   1:  PR[GP1:91,2] = PR[GP1:90,2] + -13.749;
   1:L PR[91] R[100]mm/sec CNT100;
   1:  PR[GP1:91,1] = PR[GP1:90,1] + -6.828;
   1:  PR[GP1:91,2] = PR[GP1:90,2] + -9.017;
   1:L PR[91] R[100]mm/sec CNT100;
   1:  PR[GP1:91,1] = PR[GP1:90,1] + -5.853;
   1:  PR[GP1:91,2] = PR[GP1:90,2] + -5.100;
   1:L PR[91] R[100]mm/sec CNT100;
   1:  PR[GP1:91,1] = PR[GP1:90,1] + -4.023;
   1:  PR[GP1:91,2] = PR[GP1:90,2] + -1.796;
   1:L PR[91] R[100]mm/sec CNT100;
   1:  PR[GP1:91,1] = PR[GP1:90,1] + -0.454;
   1:  PR[GP1:91,2] = PR[GP1:90,2] + -0.472;
   1:L PR[91] R[100]mm/sec CNT100;
   1:  PR[GP1:91,1] = PR[GP1:90,1] + 0.667;
   1:L PR[91] R[100]mm/sec CNT100;
   1:  PR[GP1:91,1] = PR[GP1:90,1] + 4.236;
   1:  PR[GP1:91,2] = PR[GP1:90,2] + -1.796;
   1:L PR[91] R[100]mm/sec CNT100;
   1:  PR[GP1:91,1] = PR[GP1:90,1] + 6.052;
   1:  PR[GP1:91,2] = PR[GP1:90,2] + -5.076;
   1:L PR[91] R[100]mm/sec CNT100;
   1:  PR[GP1:91,1] = PR[GP1:90,1] + 7.757;
   1:  PR[GP1:91,2] = PR[GP1:90,2] + -9.935;
   1:L PR[91] R[100]mm/sec CNT100;
   1:  PR[GP1:91,1] = PR[GP1:90,1] + 8.713;
   1:  PR[GP1:91,2] = PR[GP1:90,2] + -13.775;
   1:L PR[91] R[100]mm/sec CNT100;
   1:  PR[GP1:91,1] = PR[GP1:90,1] + 10.319;
   1:  PR[GP1:91,2] = PR[GP1:90,2] + -17.268;
   1:L PR[91] R[100]mm/sec CNT100;
   1:  PR[GP1:91,1] = PR[GP1:90,1] + 13.595;
   1:  PR[GP1:91,2] = PR[GP1:90,2] + -21.070;
   1:L PR[91] R[100]mm/sec CNT100;
   1:  PR[GP1:91,1] = PR[GP1:90,1] + 15.888;
   1:  PR[GP1:91,2] = PR[GP1:90,2] + -24.295;
   1:L PR[91] R[100]mm/sec CNT100;
   1:  PR[GP1:91,1] = PR[GP1:90,1] + 18.658;
   1:  PR[GP1:91,2] = PR[GP1:90,2] + -26.960;
   1:L PR[91] R[100]mm/sec CNT100;
   1:  PR[GP1:91,1] = PR[GP1:90,1] + 23.094;
   1:  PR[GP1:91,2] = PR[GP1:90,2] + -29.301;
   1:L PR[91] R[100]mm/sec CNT100;
   1:  PR[GP1:91,1] = PR[GP1:90,1] + 26.406;
   1:  PR[GP1:91,2] = PR[GP1:90,2] + -31.467;
   1:L PR[91] R[100]mm/sec CNT100;
   1:  PR[GP1:91,1] = PR[GP1:90,1] + 29.959;
   1:  PR[GP1:91,2] = PR[GP1:90,2] + -32.936;
   1:L PR[91] R[100]mm/sec CNT100;
   1:  PR[GP1:91,1] = PR[GP1:90,1] + 34.945;
   1:  PR[GP1:91,2] = PR[GP1:90,2] + -33.495;
   1:L PR[91] R[100]mm/sec CNT100;
   1:  PR[GP1:91,1] = PR[GP1:90,1] + 38.819;
   1:  PR[GP1:91,2] = PR[GP1:90,2] + -34.301;
   1:L PR[91] R[100]mm/sec CNT100;
   1:  PR[GP1:91,1] = PR[GP1:90,1] + 42.663;
   1:  PR[GP1:91,2] = PR[GP1:90,2] + -34.371;
   1:L PR[91] R[100]mm/sec CNT100;
   1:  PR[GP1:91,1] = PR[GP1:90,1] + 47.510;
   1:  PR[GP1:91,2] = PR[GP1:90,2] + -33.071;
   1:L PR[91] R[100]mm/sec CNT100;
   1:  PR[GP1:91,1] = PR[GP1:90,1] + 51.411;
   1:  PR[GP1:91,2] = PR[GP1:90,2] + -32.407;
   1:L PR[91] R[100]mm/sec CNT100;
   1:  PR[GP1:91,1] = PR[GP1:90,1] + 55.014;
   1:  PR[GP1:91,2] = PR[GP1:90,2] + -31.068;
   1:L PR[91] R[100]mm/sec CNT100;
   1:  PR[GP1:91,1] = PR[GP1:90,1] + 59.050;
   1:  PR[GP1:91,2] = PR[GP1:90,2] + -28.089;
   1:L PR[91] R[100]mm/sec CNT100;
   1:  PR[GP1:91,1] = PR[GP1:90,1] + 62.438;
   1:  PR[GP1:91,2] = PR[GP1:90,2] + -26.045;
   1:L PR[91] R[100]mm/sec CNT100;
   1:  PR[GP1:91,1] = PR[GP1:90,1] + 65.304;
   1:  PR[GP1:91,2] = PR[GP1:90,2] + -23.483;
   1:L PR[91] R[100]mm/sec CNT100;
   1:  PR[GP1:91,1] = PR[GP1:90,1] + 67.974;
   1:  PR[GP1:91,2] = PR[GP1:90,2] + -19.233;
   1:L PR[91] R[100]mm/sec CNT100;
   1:  PR[GP1:91,1] = PR[GP1:90,1] + 70.383;
   1:  PR[GP1:91,2] = PR[GP1:90,2] + -16.093;
   1:L PR[91] R[100]mm/sec CNT100;
   1:  PR[GP1:91,1] = PR[GP1:90,1] + 72.115;
   1:  PR[GP1:91,2] = PR[GP1:90,2] + -12.661;
   1:L PR[91] R[100]mm/sec CNT100;
   1:  PR[GP1:91,1] = PR[GP1:90,1] + 73.047;
   1:  PR[GP1:91,2] = PR[GP1:90,2] + -7.730;
   1:L PR[91] R[100]mm/sec CNT100;
   1:  PR[GP1:91,1] = PR[GP1:90,1] + 74.143;
   1:  PR[GP1:91,2] = PR[GP1:90,2] + -3.928;
   1:L PR[91] R[100]mm/sec CNT100;
   1:  PR[GP1:91,1] = PR[GP1:90,1] + 74.501;
   1:  PR[GP1:91,2] = PR[GP1:90,2] + -0.100;
   1:L PR[91] R[100]mm/sec CNT100;
   1:  PR[GP1:91,1] = PR[GP1:90,1] + 73.568;
   1:  PR[GP1:91,2] = PR[GP1:90,2] + 4.830;
   1:L PR[91] R[100]mm/sec CNT100;
   1:  PR[GP1:91,1] = PR[GP1:90,1] + 73.199;
   1:  PR[GP1:91,2] = PR[GP1:90,2] + 8.770;
   1:L PR[91] R[100]mm/sec CNT100;
   1:  PR[GP1:91,1] = PR[GP1:90,1] + 72.127;
   1:  PR[GP1:91,2] = PR[GP1:90,2] + 12.491;
   1:L PR[91] R[100]mm/sec CNT100;
   1:  PR[GP1:91,1] = PR[GP1:90,1] + 70.370;
   1:  PR[GP1:91,2] = PR[GP1:90,2] + 15.974;
   1:L PR[91] R[100]mm/sec CNT100;
   1:  PR[GP1:91,1] = PR[GP1:90,1] + 67.700;
   1:  PR[GP1:91,2] = PR[GP1:90,2] + 20.225;
   1:L PR[91] R[100]mm/sec CNT100;
   1:  PR[GP1:91,1] = PR[GP1:90,1] + 65.325;
   1:  PR[GP1:91,2] = PR[GP1:90,2] + 23.320;
   1:L PR[91] R[100]mm/sec CNT100;
   1:  PR[GP1:91,1] = PR[GP1:90,1] + 62.417;
   1:  PR[GP1:91,2] = PR[GP1:90,2] + 25.920;
   1:L PR[91] R[100]mm/sec CNT100;
   1:  PR[GP1:91,1] = PR[GP1:90,1] + 58.382;
   1:  PR[GP1:91,2] = PR[GP1:90,2] + 28.900;
   1:L PR[91] R[100]mm/sec CNT100;
   1:  PR[GP1:91,1] = PR[GP1:90,1] + 55.041;
   1:  PR[GP1:91,2] = PR[GP1:90,2] + 30.914;
   1:L PR[91] R[100]mm/sec CNT100;
   1:  PR[GP1:91,1] = PR[GP1:90,1] + 51.384;
   1:  PR[GP1:91,2] = PR[GP1:90,2] + 32.273;
   1:L PR[91] R[100]mm/sec CNT100;
   1:  PR[GP1:91,1] = PR[GP1:90,1] + 46.537;
   1:  PR[GP1:91,2] = PR[GP1:90,2] + 33.573;
   1:L PR[91] R[100]mm/sec CNT100;
   1:  PR[GP1:91,1] = PR[GP1:90,1] + 42.691;
   1:  PR[GP1:91,2] = PR[GP1:90,2] + 34.228;
   1:L PR[91] R[100]mm/sec CNT100;
   1:  PR[GP1:91,1] = PR[GP1:90,1] + 38.791;
   1:  PR[GP1:91,2] = PR[GP1:90,2] + 34.157;
   1:L PR[91] R[100]mm/sec CNT100;
   1:  PR[GP1:91,1] = PR[GP1:90,1] + 33.804;
   1:  PR[GP1:91,2] = PR[GP1:90,2] + 33.597;
   1:L PR[91] R[100]mm/sec CNT100;
   1:  PR[GP1:91,1] = PR[GP1:90,1] + 29.985;
   1:  PR[GP1:91,2] = PR[GP1:90,2] + 32.802;
   1:L PR[91] R[100]mm/sec CNT100;
   1:  PR[GP1:91,1] = PR[GP1:90,1] + 26.380;
   1:  PR[GP1:91,2] = PR[GP1:90,2] + 31.312;
   1:L PR[91] R[100]mm/sec CNT100;
   1:  PR[GP1:91,1] = PR[GP1:90,1] + 21.944;
   1:  PR[GP1:91,2] = PR[GP1:90,2] + 28.970;
   1:L PR[91] R[100]mm/sec CNT100;
   1:  PR[GP1:91,1] = PR[GP1:90,1] + 18.679;
   1:  PR[GP1:91,2] = PR[GP1:90,2] + 26.836;
   1:L PR[91] R[100]mm/sec CNT100;
   1:  PR[GP1:91,1] = PR[GP1:90,1] + 15.867;
   1:  PR[GP1:91,2] = PR[GP1:90,2] + 24.131;
   1:L PR[91] R[100]mm/sec CNT100;
   1:  PR[GP1:91,1] = PR[GP1:90,1] + 12.591;
   1:  PR[GP1:91,2] = PR[GP1:90,2] + 20.329;
   1:L PR[91] R[100]mm/sec CNT100;
   1:  PR[GP1:91,1] = PR[GP1:90,1] + 10.331;
   1:  PR[GP1:91,2] = PR[GP1:90,2] + 17.150;
   1:L PR[91] R[100]mm/sec CNT100;
   1:  PR[GP1:91,1] = PR[GP1:90,1] + 8.701;
   1:  PR[GP1:91,2] = PR[GP1:90,2] + 13.605;
   1:L PR[91] R[100]mm/sec CNT100;
   1:  PR[GP1:91,1] = PR[GP1:90,1] + 7.041;
   1:  PR[GP1:91,2] = PR[GP1:90,2] + 8.873;
   1:L PR[91] R[100]mm/sec CNT100;
   1:  PR[GP1:91,1] = PR[GP1:90,1] + 6.066;
   1:  PR[GP1:91,2] = PR[GP1:90,2] + 4.956;
   1:L PR[91] R[100]mm/sec CNT100;
   1:  PR[GP1:91,1] = PR[GP1:90,1] + 4.236;
   1:  PR[GP1:91,2] = PR[GP1:90,2] + 1.652;
   1:L PR[91] R[100]mm/sec CNT100;
   1:  PR[GP1:91,1] = PR[GP1:90,1] + 0.667;
   1:  PR[GP1:91,2] = PR[GP1:90,2] + 0.328;
   1:L PR[91] R[100]mm/sec CNT100;
   1:  PR[GP1:91,1] = PR[GP1:90,1] + -0.454;
   1:L PR[91] R[100]mm/sec CNT100;
   1:  ! -- Layer/Ebene 9 -- !;
   1:  PR[91] = PR[90];
   1:  PR[GP1:91,1] = PR[GP1:90,1] + -4.023;
   1:  PR[GP1:91,2] = PR[GP1:90,2] + 1.652;
   1:  PR[GP1:91,3] = PR[GP1:90,3] + 5.795;
   1:L PR[91] R[100]mm/sec CNT100;
   1:  PR[GP1:91,1] = PR[GP1:90,1] + -5.839;
   1:  PR[GP1:91,2] = PR[GP1:90,2] + 4.932;
   1:L PR[91] R[100]mm/sec CNT100;
   1:  PR[GP1:91,1] = PR[GP1:90,1] + -7.216;
   1:  PR[GP1:91,2] = PR[GP1:90,2] + 8.855;
   1:L PR[91] R[100]mm/sec CNT100;
   1:  PR[GP1:91,1] = PR[GP1:90,1] + -8.292;
   1:  PR[GP1:91,2] = PR[GP1:90,2] + 13.179;
   1:L PR[91] R[100]mm/sec CNT100;
   1:  PR[GP1:91,1] = PR[GP1:90,1] + -10.106;
   1:  PR[GP1:91,2] = PR[GP1:90,2] + 17.124;
   1:L PR[91] R[100]mm/sec CNT100;
   1:  PR[GP1:91,1] = PR[GP1:90,1] + -12.734;
   1:  PR[GP1:91,2] = PR[GP1:90,2] + 20.174;
   1:L PR[91] R[100]mm/sec CNT100;
   1:  PR[GP1:91,1] = PR[GP1:90,1] + -15.315;
   1:  PR[GP1:91,2] = PR[GP1:90,2] + 23.806;
   1:L PR[91] R[100]mm/sec CNT100;
   1:  PR[GP1:91,1] = PR[GP1:90,1] + -18.445;
   1:  PR[GP1:91,2] = PR[GP1:90,2] + 26.816;
   1:L PR[91] R[100]mm/sec CNT100;
   1:  PR[GP1:91,1] = PR[GP1:90,1] + -22.004;
   1:  PR[GP1:91,2] = PR[GP1:90,2] + 28.695;
   1:L PR[91] R[100]mm/sec CNT100;
   1:  PR[GP1:91,1] = PR[GP1:90,1] + -25.733;
   1:  PR[GP1:91,2] = PR[GP1:90,2] + 31.132;
   1:L PR[91] R[100]mm/sec CNT100;
   1:  PR[GP1:91,1] = PR[GP1:90,1] + -29.746;
   1:  PR[GP1:91,2] = PR[GP1:90,2] + 32.792;
   1:L PR[91] R[100]mm/sec CNT100;
   1:  PR[GP1:91,1] = PR[GP1:90,1] + -33.747;
   1:  PR[GP1:91,2] = PR[GP1:90,2] + 33.241;
   1:L PR[91] R[100]mm/sec CNT100;
   1:  PR[GP1:91,1] = PR[GP1:90,1] + -38.108;
   1:  PR[GP1:91,2] = PR[GP1:90,2] + 34.148;
   1:L PR[91] R[100]mm/sec CNT100;
   1:  PR[GP1:91,1] = PR[GP1:90,1] + -42.450;
   1:  PR[GP1:91,2] = PR[GP1:90,2] + 34.227;
   1:L PR[91] R[100]mm/sec CNT100;
   1:  PR[GP1:91,1] = PR[GP1:90,1] + -46.339;
   1:  PR[GP1:91,2] = PR[GP1:90,2] + 33.184;
   1:L PR[91] R[100]mm/sec CNT100;
   1:  PR[GP1:91,1] = PR[GP1:90,1] + -50.731;
   1:  PR[GP1:91,2] = PR[GP1:90,2] + 32.436;
   1:L PR[91] R[100]mm/sec CNT100;
   1:  PR[GP1:91,1] = PR[GP1:90,1] + -54.801;
   1:  PR[GP1:91,2] = PR[GP1:90,2] + 30.924;
   1:L PR[91] R[100]mm/sec CNT100;
   1:  PR[GP1:91,1] = PR[GP1:90,1] + -58.039;
   1:  PR[GP1:91,2] = PR[GP1:90,2] + 28.534;
   1:L PR[91] R[100]mm/sec CNT100;
   1:  PR[GP1:91,1] = PR[GP1:90,1] + -61.854;
   1:  PR[GP1:91,2] = PR[GP1:90,2] + 26.233;
   1:L PR[91] R[100]mm/sec CNT100;
   1:  PR[GP1:91,1] = PR[GP1:90,1] + -65.091;
   1:  PR[GP1:91,2] = PR[GP1:90,2] + 23.338;
   1:L PR[91] R[100]mm/sec CNT100;
   1:  PR[GP1:91,1] = PR[GP1:90,1] + -67.234;
   1:  PR[GP1:91,2] = PR[GP1:90,2] + 19.929;
   1:L PR[91] R[100]mm/sec CNT100;
   1:  PR[GP1:91,1] = PR[GP1:90,1] + -69.945;
   1:  PR[GP1:91,2] = PR[GP1:90,2] + 16.394;
   1:L PR[91] R[100]mm/sec CNT100;
   1:  PR[GP1:91,1] = PR[GP1:90,1] + -71.901;
   1:  PR[GP1:91,2] = PR[GP1:90,2] + 12.517;
   1:L PR[91] R[100]mm/sec CNT100;
   1:  PR[GP1:91,1] = PR[GP1:90,1] + -72.650;
   1:  PR[GP1:91,2] = PR[GP1:90,2] + 8.561;
   1:L PR[91] R[100]mm/sec CNT100;
   1:  PR[GP1:91,1] = PR[GP1:90,1] + -73.883;
   1:  PR[GP1:91,2] = PR[GP1:90,2] + 4.280;
   1:L PR[91] R[100]mm/sec CNT100;
   1:  PR[GP1:91,1] = PR[GP1:90,1] + -74.288;
   1:  PR[GP1:91,2] = PR[GP1:90,2] + -0.044;
   1:L PR[91] R[100]mm/sec CNT100;
   1:  PR[GP1:91,1] = PR[GP1:90,1] + -73.540;
   1:  PR[GP1:91,2] = PR[GP1:90,2] + -3.999;
   1:L PR[91] R[100]mm/sec CNT100;
   1:  PR[GP1:91,1] = PR[GP1:90,1] + -73.124;
   1:  PR[GP1:91,2] = PR[GP1:90,2] + -8.435;
   1:L PR[91] R[100]mm/sec CNT100;
   1:  PR[GP1:91,1] = PR[GP1:90,1] + -71.914;
   1:  PR[GP1:91,2] = PR[GP1:90,2] + -12.635;
   1:L PR[91] R[100]mm/sec CNT100;
   1:  PR[GP1:91,1] = PR[GP1:90,1] + -69.932;
   1:  PR[GP1:91,2] = PR[GP1:90,2] + -16.563;
   1:L PR[91] R[100]mm/sec CNT100;
   1:  PR[GP1:91,1] = PR[GP1:90,1] + -67.790;
   1:  PR[GP1:91,2] = PR[GP1:90,2] + -19.973;
   1:L PR[91] R[100]mm/sec CNT100;
   1:  PR[GP1:91,1] = PR[GP1:90,1] + -65.113;
   1:  PR[GP1:91,2] = PR[GP1:90,2] + -23.464;
   1:L PR[91] R[100]mm/sec CNT100;
   1:  PR[GP1:91,1] = PR[GP1:90,1] + -61.833;
   1:  PR[GP1:91,2] = PR[GP1:90,2] + -26.396;
   1:L PR[91] R[100]mm/sec CNT100;
   1:  PR[GP1:91,1] = PR[GP1:90,1] + -58.595;
   1:  PR[GP1:91,2] = PR[GP1:90,2] + -28.786;
   1:L PR[91] R[100]mm/sec CNT100;
   1:  PR[GP1:91,1] = PR[GP1:90,1] + -54.828;
   1:  PR[GP1:91,2] = PR[GP1:90,2] + -31.058;
   1:L PR[91] R[100]mm/sec CNT100;
   1:  PR[GP1:91,1] = PR[GP1:90,1] + -50.704;
   1:  PR[GP1:91,2] = PR[GP1:90,2] + -32.590;
   1:L PR[91] R[100]mm/sec CNT100;
   1:  PR[GP1:91,1] = PR[GP1:90,1] + -46.815;
   1:  PR[GP1:91,2] = PR[GP1:90,2] + -33.633;
   1:L PR[91] R[100]mm/sec CNT100;
   1:  PR[GP1:91,1] = PR[GP1:90,1] + -42.479;
   1:  PR[GP1:91,2] = PR[GP1:90,2] + -34.372;
   1:L PR[91] R[100]mm/sec CNT100;
   1:  PR[GP1:91,1] = PR[GP1:90,1] + -38.080;
   1:  PR[GP1:91,2] = PR[GP1:90,2] + -34.292;
   1:L PR[91] R[100]mm/sec CNT100;
   1:  PR[GP1:91,1] = PR[GP1:90,1] + -34.079;
   1:  PR[GP1:91,2] = PR[GP1:90,2] + -33.843;
   1:L PR[91] R[100]mm/sec CNT100;
   1:  PR[GP1:91,1] = PR[GP1:90,1] + -29.772;
   1:  PR[GP1:91,2] = PR[GP1:90,2] + -32.947;
   1:L PR[91] R[100]mm/sec CNT100;
   1:  PR[GP1:91,1] = PR[GP1:90,1] + -25.707;
   1:  PR[GP1:91,2] = PR[GP1:90,2] + -31.266;
   1:L PR[91] R[100]mm/sec CNT100;
   1:  PR[GP1:91,1] = PR[GP1:90,1] + -22.148;
   1:  PR[GP1:91,2] = PR[GP1:90,2] + -29.387;
   1:L PR[91] R[100]mm/sec CNT100;
   1:  PR[GP1:91,1] = PR[GP1:90,1] + -18.466;
   1:  PR[GP1:91,2] = PR[GP1:90,2] + -26.980;
   1:L PR[91] R[100]mm/sec CNT100;
   1:  PR[GP1:91,1] = PR[GP1:90,1] + -15.295;
   1:  PR[GP1:91,2] = PR[GP1:90,2] + -23.930;
   1:L PR[91] R[100]mm/sec CNT100;
   1:  PR[GP1:91,1] = PR[GP1:90,1] + -12.667;
   1:  PR[GP1:91,2] = PR[GP1:90,2] + -20.880;
   1:L PR[91] R[100]mm/sec CNT100;
   1:  PR[GP1:91,1] = PR[GP1:90,1] + -10.118;
   1:  PR[GP1:91,2] = PR[GP1:90,2] + -17.294;
   1:L PR[91] R[100]mm/sec CNT100;
   1:  PR[GP1:91,1] = PR[GP1:90,1] + -8.280;
   1:  PR[GP1:91,2] = PR[GP1:90,2] + -13.297;
   1:L PR[91] R[100]mm/sec CNT100;
   1:  PR[GP1:91,1] = PR[GP1:90,1] + -6.948;
   1:  PR[GP1:91,2] = PR[GP1:90,2] + -9.500;
   1:L PR[91] R[100]mm/sec CNT100;
   1:  PR[GP1:91,1] = PR[GP1:90,1] + -5.853;
   1:  PR[GP1:91,2] = PR[GP1:90,2] + -5.100;
   1:L PR[91] R[100]mm/sec CNT100;
   1:  PR[GP1:91,1] = PR[GP1:90,1] + -4.023;
   1:  PR[GP1:91,2] = PR[GP1:90,2] + -1.795;
   1:L PR[91] R[100]mm/sec CNT100;
   1:  PR[GP1:91,1] = PR[GP1:90,1] + -0.454;
   1:  PR[GP1:91,2] = PR[GP1:90,2] + -0.472;
   1:L PR[91] R[100]mm/sec CNT100;
   1:  PR[GP1:91,1] = PR[GP1:90,1] + 0.667;
   1:L PR[91] R[100]mm/sec CNT100;
   1:  PR[GP1:91,1] = PR[GP1:90,1] + 4.236;
   1:  PR[GP1:91,2] = PR[GP1:90,2] + -1.795;
   1:L PR[91] R[100]mm/sec CNT100;
   1:  PR[GP1:91,1] = PR[GP1:90,1] + 6.052;
   1:  PR[GP1:91,2] = PR[GP1:90,2] + -5.076;
   1:L PR[91] R[100]mm/sec CNT100;
   1:  PR[GP1:91,1] = PR[GP1:90,1] + 7.429;
   1:  PR[GP1:91,2] = PR[GP1:90,2] + -9.000;
   1:L PR[91] R[100]mm/sec CNT100;
   1:  PR[GP1:91,1] = PR[GP1:90,1] + 8.505;
   1:  PR[GP1:91,2] = PR[GP1:90,2] + -13.323;
   1:L PR[91] R[100]mm/sec CNT100;
   1:  PR[GP1:91,1] = PR[GP1:90,1] + 10.319;
   1:  PR[GP1:91,2] = PR[GP1:90,2] + -17.268;
   1:L PR[91] R[100]mm/sec CNT100;
   1:  PR[GP1:91,1] = PR[GP1:90,1] + 12.948;
   1:  PR[GP1:91,2] = PR[GP1:90,2] + -20.318;
   1:L PR[91] R[100]mm/sec CNT100;
   1:  PR[GP1:91,1] = PR[GP1:90,1] + 15.529;
   1:  PR[GP1:91,2] = PR[GP1:90,2] + -23.950;
   1:L PR[91] R[100]mm/sec CNT100;
   1:  PR[GP1:91,1] = PR[GP1:90,1] + 18.659;
   1:  PR[GP1:91,2] = PR[GP1:90,2] + -26.960;
   1:L PR[91] R[100]mm/sec CNT100;
   1:  PR[GP1:91,1] = PR[GP1:90,1] + 22.217;
   1:  PR[GP1:91,2] = PR[GP1:90,2] + -28.839;
   1:L PR[91] R[100]mm/sec CNT100;
   1:  PR[GP1:91,1] = PR[GP1:90,1] + 25.946;
   1:  PR[GP1:91,2] = PR[GP1:90,2] + -31.276;
   1:L PR[91] R[100]mm/sec CNT100;
   1:  PR[GP1:91,1] = PR[GP1:90,1] + 29.959;
   1:  PR[GP1:91,2] = PR[GP1:90,2] + -32.936;
   1:L PR[91] R[100]mm/sec CNT100;
   1:  PR[GP1:91,1] = PR[GP1:90,1] + 33.960;
   1:  PR[GP1:91,2] = PR[GP1:90,2] + -33.385;
   1:L PR[91] R[100]mm/sec CNT100;
   1:  PR[GP1:91,1] = PR[GP1:90,1] + 38.322;
   1:  PR[GP1:91,2] = PR[GP1:90,2] + -34.292;
   1:L PR[91] R[100]mm/sec CNT100;
   1:  PR[GP1:91,1] = PR[GP1:90,1] + 42.663;
   1:  PR[GP1:91,2] = PR[GP1:90,2] + -34.371;
   1:L PR[91] R[100]mm/sec CNT100;
   1:  PR[GP1:91,1] = PR[GP1:90,1] + 46.552;
   1:  PR[GP1:91,2] = PR[GP1:90,2] + -33.328;
   1:L PR[91] R[100]mm/sec CNT100;
   1:  PR[GP1:91,1] = PR[GP1:90,1] + 50.944;
   1:  PR[GP1:91,2] = PR[GP1:90,2] + -32.580;
   1:L PR[91] R[100]mm/sec CNT100;
   1:  PR[GP1:91,1] = PR[GP1:90,1] + 55.015;
   1:  PR[GP1:91,2] = PR[GP1:90,2] + -31.068;
   1:L PR[91] R[100]mm/sec CNT100;
   1:  PR[GP1:91,1] = PR[GP1:90,1] + 58.252;
   1:  PR[GP1:91,2] = PR[GP1:90,2] + -28.678;
   1:L PR[91] R[100]mm/sec CNT100;
   1:  PR[GP1:91,1] = PR[GP1:90,1] + 62.067;
   1:  PR[GP1:91,2] = PR[GP1:90,2] + -26.377;
   1:L PR[91] R[100]mm/sec CNT100;
   1:  PR[GP1:91,1] = PR[GP1:90,1] + 65.305;
   1:  PR[GP1:91,2] = PR[GP1:90,2] + -23.482;
   1:L PR[91] R[100]mm/sec CNT100;
   1:  PR[GP1:91,1] = PR[GP1:90,1] + 67.447;
   1:  PR[GP1:91,2] = PR[GP1:90,2] + -20.073;
   1:L PR[91] R[100]mm/sec CNT100;
   1:  PR[GP1:91,1] = PR[GP1:90,1] + 70.158;
   1:  PR[GP1:91,2] = PR[GP1:90,2] + -16.538;
   1:L PR[91] R[100]mm/sec CNT100;
   1:  PR[GP1:91,1] = PR[GP1:90,1] + 72.115;
   1:  PR[GP1:91,2] = PR[GP1:90,2] + -12.661;
   1:L PR[91] R[100]mm/sec CNT100;
   1:  PR[GP1:91,1] = PR[GP1:90,1] + 72.863;
   1:  PR[GP1:91,2] = PR[GP1:90,2] + -8.705;
   1:L PR[91] R[100]mm/sec CNT100;
   1:  PR[GP1:91,1] = PR[GP1:90,1] + 74.096;
   1:  PR[GP1:91,2] = PR[GP1:90,2] + -4.424;
   1:L PR[91] R[100]mm/sec CNT100;
   1:  PR[GP1:91,1] = PR[GP1:90,1] + 74.501;
   1:  PR[GP1:91,2] = PR[GP1:90,2] + -0.100;
   1:L PR[91] R[100]mm/sec CNT100;
   1:  PR[GP1:91,1] = PR[GP1:90,1] + 73.753;
   1:  PR[GP1:91,2] = PR[GP1:90,2] + 3.855;
   1:L PR[91] R[100]mm/sec CNT100;
   1:  PR[GP1:91,1] = PR[GP1:90,1] + 73.337;
   1:  PR[GP1:91,2] = PR[GP1:90,2] + 8.291;
   1:L PR[91] R[100]mm/sec CNT100;
   1:  PR[GP1:91,1] = PR[GP1:90,1] + 72.127;
   1:  PR[GP1:91,2] = PR[GP1:90,2] + 12.491;
   1:L PR[91] R[100]mm/sec CNT100;
   1:  PR[GP1:91,1] = PR[GP1:90,1] + 70.145;
   1:  PR[GP1:91,2] = PR[GP1:90,2] + 16.419;
   1:L PR[91] R[100]mm/sec CNT100;
   1:  PR[GP1:91,1] = PR[GP1:90,1] + 68.003;
   1:  PR[GP1:91,2] = PR[GP1:90,2] + 19.829;
   1:L PR[91] R[100]mm/sec CNT100;
   1:  PR[GP1:91,1] = PR[GP1:90,1] + 65.326;
   1:  PR[GP1:91,2] = PR[GP1:90,2] + 23.320;
   1:L PR[91] R[100]mm/sec CNT100;
   1:  PR[GP1:91,1] = PR[GP1:90,1] + 62.046;
   1:  PR[GP1:91,2] = PR[GP1:90,2] + 26.252;
   1:L PR[91] R[100]mm/sec CNT100;
   1:  PR[GP1:91,1] = PR[GP1:90,1] + 58.809;
   1:  PR[GP1:91,2] = PR[GP1:90,2] + 28.642;
   1:L PR[91] R[100]mm/sec CNT100;
   1:  PR[GP1:91,1] = PR[GP1:90,1] + 55.041;
   1:  PR[GP1:91,2] = PR[GP1:90,2] + 30.914;
   1:L PR[91] R[100]mm/sec CNT100;
   1:  PR[GP1:91,1] = PR[GP1:90,1] + 50.917;
   1:  PR[GP1:91,2] = PR[GP1:90,2] + 32.446;
   1:L PR[91] R[100]mm/sec CNT100;
   1:  PR[GP1:91,1] = PR[GP1:90,1] + 47.029;
   1:  PR[GP1:91,2] = PR[GP1:90,2] + 33.489;
   1:L PR[91] R[100]mm/sec CNT100;
   1:  PR[GP1:91,1] = PR[GP1:90,1] + 42.692;
   1:  PR[GP1:91,2] = PR[GP1:90,2] + 34.228;
   1:L PR[91] R[100]mm/sec CNT100;
   1:  PR[GP1:91,1] = PR[GP1:90,1] + 38.293;
   1:  PR[GP1:91,2] = PR[GP1:90,2] + 34.148;
   1:L PR[91] R[100]mm/sec CNT100;
   1:  PR[GP1:91,1] = PR[GP1:90,1] + 34.292;
   1:  PR[GP1:91,2] = PR[GP1:90,2] + 33.699;
   1:L PR[91] R[100]mm/sec CNT100;
   1:  PR[GP1:91,1] = PR[GP1:90,1] + 29.985;
   1:  PR[GP1:91,2] = PR[GP1:90,2] + 32.803;
   1:L PR[91] R[100]mm/sec CNT100;
   1:  PR[GP1:91,1] = PR[GP1:90,1] + 25.920;
   1:  PR[GP1:91,2] = PR[GP1:90,2] + 31.122;
   1:L PR[91] R[100]mm/sec CNT100;
   1:  PR[GP1:91,1] = PR[GP1:90,1] + 22.361;
   1:  PR[GP1:91,2] = PR[GP1:90,2] + 29.243;
   1:L PR[91] R[100]mm/sec CNT100;
   1:  PR[GP1:91,1] = PR[GP1:90,1] + 18.679;
   1:  PR[GP1:91,2] = PR[GP1:90,2] + 26.836;
   1:L PR[91] R[100]mm/sec CNT100;
   1:  PR[GP1:91,1] = PR[GP1:90,1] + 15.508;
   1:  PR[GP1:91,2] = PR[GP1:90,2] + 23.786;
   1:L PR[91] R[100]mm/sec CNT100;
   1:  PR[GP1:91,1] = PR[GP1:90,1] + 12.880;
   1:  PR[GP1:91,2] = PR[GP1:90,2] + 20.736;
   1:L PR[91] R[100]mm/sec CNT100;
   1:  PR[GP1:91,1] = PR[GP1:90,1] + 10.331;
   1:  PR[GP1:91,2] = PR[GP1:90,2] + 17.150;
   1:L PR[91] R[100]mm/sec CNT100;
   1:  PR[GP1:91,1] = PR[GP1:90,1] + 8.494;
   1:  PR[GP1:91,2] = PR[GP1:90,2] + 13.153;
   1:L PR[91] R[100]mm/sec CNT100;
   1:  PR[GP1:91,1] = PR[GP1:90,1] + 7.161;
   1:  PR[GP1:91,2] = PR[GP1:90,2] + 9.356;
   1:L PR[91] R[100]mm/sec CNT100;
   1:  PR[GP1:91,1] = PR[GP1:90,1] + 6.066;
   1:  PR[GP1:91,2] = PR[GP1:90,2] + 4.956;
   1:L PR[91] R[100]mm/sec CNT100;
   1:  PR[GP1:91,1] = PR[GP1:90,1] + 4.236;
   1:  PR[GP1:91,2] = PR[GP1:90,2] + 1.652;
   1:L PR[91] R[100]mm/sec CNT100;
   1:  PR[GP1:91,1] = PR[GP1:90,1] + 0.667;
   1:  PR[GP1:91,2] = PR[GP1:90,2] + 0.328;
   1:L PR[91] R[100]mm/sec CNT100;
   1:  PR[GP1:91,1] = PR[GP1:90,1] + -0.454;
   1:L PR[91] R[100]mm/sec CNT100;
   1:  ! -- Layer/Ebene 10 -- !;
   1:  PR[91] = PR[90];
   1:  PR[GP1:91,1] = PR[GP1:90,1] + -4.023;
   1:  PR[GP1:91,2] = PR[GP1:90,2] + 1.651;
   1:  PR[GP1:91,3] = PR[GP1:90,3] + 6.405;
   1:L PR[91] R[100]mm/sec CNT100;
   1:  PR[GP1:91,1] = PR[GP1:90,1] + -5.839;
   1:  PR[GP1:91,2] = PR[GP1:90,2] + 4.932;
   1:L PR[91] R[100]mm/sec CNT100;
   1:  PR[GP1:91,1] = PR[GP1:90,1] + -6.887;
   1:  PR[GP1:91,2] = PR[GP1:90,2] + 7.920;
   1:L PR[91] R[100]mm/sec CNT100;
   1:  PR[GP1:91,1] = PR[GP1:90,1] + -8.084;
   1:  PR[GP1:91,2] = PR[GP1:90,2] + 12.727;
   1:L PR[91] R[100]mm/sec CNT100;
   1:  PR[GP1:91,1] = PR[GP1:90,1] + -10.106;
   1:  PR[GP1:91,2] = PR[GP1:90,2] + 17.125;
   1:L PR[91] R[100]mm/sec CNT100;
   1:  PR[GP1:91,1] = PR[GP1:90,1] + -12.087;
   1:  PR[GP1:91,2] = PR[GP1:90,2] + 19.423;
   1:L PR[91] R[100]mm/sec CNT100;
   1:  PR[GP1:91,1] = PR[GP1:90,1] + -14.957;
   1:  PR[GP1:91,2] = PR[GP1:90,2] + 23.461;
   1:L PR[91] R[100]mm/sec CNT100;
   1:  PR[GP1:91,1] = PR[GP1:90,1] + -18.445;
   1:  PR[GP1:91,2] = PR[GP1:90,2] + 26.816;
   1:L PR[91] R[100]mm/sec CNT100;
   1:  PR[GP1:91,1] = PR[GP1:90,1] + -21.127;
   1:  PR[GP1:91,2] = PR[GP1:90,2] + 28.232;
   1:L PR[91] R[100]mm/sec CNT100;
   1:  PR[GP1:91,1] = PR[GP1:90,1] + -25.273;
   1:  PR[GP1:91,2] = PR[GP1:90,2] + 30.942;
   1:L PR[91] R[100]mm/sec CNT100;
   1:  PR[GP1:91,1] = PR[GP1:90,1] + -29.747;
   1:  PR[GP1:91,2] = PR[GP1:90,2] + 32.792;
   1:L PR[91] R[100]mm/sec CNT100;
   1:  PR[GP1:91,1] = PR[GP1:90,1] + -32.761;
   1:  PR[GP1:91,2] = PR[GP1:90,2] + 33.130;
   1:L PR[91] R[100]mm/sec CNT100;
   1:  PR[GP1:91,1] = PR[GP1:90,1] + -37.611;
   1:  PR[GP1:91,2] = PR[GP1:90,2] + 34.139;
   1:L PR[91] R[100]mm/sec CNT100;
   1:  PR[GP1:91,1] = PR[GP1:90,1] + -42.451;
   1:  PR[GP1:91,2] = PR[GP1:90,2] + 34.227;
   1:L PR[91] R[100]mm/sec CNT100;
   1:  PR[GP1:91,1] = PR[GP1:90,1] + -45.381;
   1:  PR[GP1:91,2] = PR[GP1:90,2] + 33.441;
   1:L PR[91] R[100]mm/sec CNT100;
   1:  PR[GP1:91,1] = PR[GP1:90,1] + -50.264;
   1:  PR[GP1:91,2] = PR[GP1:90,2] + 32.610;
   1:L PR[91] R[100]mm/sec CNT100;
   1:  PR[GP1:91,1] = PR[GP1:90,1] + -54.802;
   1:  PR[GP1:91,2] = PR[GP1:90,2] + 30.924;
   1:L PR[91] R[100]mm/sec CNT100;
   1:  PR[GP1:91,1] = PR[GP1:90,1] + -57.241;
   1:  PR[GP1:91,2] = PR[GP1:90,2] + 29.123;
   1:L PR[91] R[100]mm/sec CNT100;
   1:  PR[GP1:91,1] = PR[GP1:90,1] + -61.483;
   1:  PR[GP1:91,2] = PR[GP1:90,2] + 26.565;
   1:L PR[91] R[100]mm/sec CNT100;
   1:  PR[GP1:91,1] = PR[GP1:90,1] + -65.092;
   1:  PR[GP1:91,2] = PR[GP1:90,2] + 23.338;
   1:L PR[91] R[100]mm/sec CNT100;
   1:  PR[GP1:91,1] = PR[GP1:90,1] + -66.706;
   1:  PR[GP1:91,2] = PR[GP1:90,2] + 20.769;
   1:L PR[91] R[100]mm/sec CNT100;
   1:  PR[GP1:91,1] = PR[GP1:90,1] + -69.721;
   1:  PR[GP1:91,2] = PR[GP1:90,2] + 16.838;
   1:L PR[91] R[100]mm/sec CNT100;
   1:  PR[GP1:91,1] = PR[GP1:90,1] + -71.901;
   1:  PR[GP1:91,2] = PR[GP1:90,2] + 12.517;
   1:L PR[91] R[100]mm/sec CNT100;
   1:  PR[GP1:91,1] = PR[GP1:90,1] + -72.465;
   1:  PR[GP1:91,2] = PR[GP1:90,2] + 9.536;
   1:L PR[91] R[100]mm/sec CNT100;
   1:  PR[GP1:91,1] = PR[GP1:90,1] + -73.836;
   1:  PR[GP1:91,2] = PR[GP1:90,2] + 4.776;
   1:L PR[91] R[100]mm/sec CNT100;
   1:  PR[GP1:91,1] = PR[GP1:90,1] + -74.288;
   1:  PR[GP1:91,2] = PR[GP1:90,2] + -0.044;
   1:L PR[91] R[100]mm/sec CNT100;
   1:  PR[GP1:91,1] = PR[GP1:90,1] + -73.724;
   1:  PR[GP1:91,2] = PR[GP1:90,2] + -3.024;
   1:L PR[91] R[100]mm/sec CNT100;
   1:  PR[GP1:91,1] = PR[GP1:90,1] + -73.262;
   1:  PR[GP1:91,2] = PR[GP1:90,2] + -7.956;
   1:L PR[91] R[100]mm/sec CNT100;
   1:  PR[GP1:91,1] = PR[GP1:90,1] + -71.914;
   1:  PR[GP1:91,2] = PR[GP1:90,2] + -12.635;
   1:L PR[91] R[100]mm/sec CNT100;
   1:  PR[GP1:91,1] = PR[GP1:90,1] + -69.708;
   1:  PR[GP1:91,2] = PR[GP1:90,2] + -17.007;
   1:L PR[91] R[100]mm/sec CNT100;
   1:  PR[GP1:91,1] = PR[GP1:90,1] + -68.093;
   1:  PR[GP1:91,2] = PR[GP1:90,2] + -19.577;
   1:L PR[91] R[100]mm/sec CNT100;
   1:  PR[GP1:91,1] = PR[GP1:90,1] + -65.113;
   1:  PR[GP1:91,2] = PR[GP1:90,2] + -23.463;
   1:L PR[91] R[100]mm/sec CNT100;
   1:  PR[GP1:91,1] = PR[GP1:90,1] + -61.462;
   1:  PR[GP1:91,2] = PR[GP1:90,2] + -26.728;
   1:L PR[91] R[100]mm/sec CNT100;
   1:  PR[GP1:91,1] = PR[GP1:90,1] + -59.022;
   1:  PR[GP1:91,2] = PR[GP1:90,2] + -28.529;
   1:L PR[91] R[100]mm/sec CNT100;
   1:  PR[GP1:91,1] = PR[GP1:90,1] + -54.828;
   1:  PR[GP1:91,2] = PR[GP1:90,2] + -31.058;
   1:L PR[91] R[100]mm/sec CNT100;
   1:  PR[GP1:91,1] = PR[GP1:90,1] + -50.238;
   1:  PR[GP1:91,2] = PR[GP1:90,2] + -32.763;
   1:L PR[91] R[100]mm/sec CNT100;
   1:  PR[GP1:91,1] = PR[GP1:90,1] + -47.307;
   1:  PR[GP1:91,2] = PR[GP1:90,2] + -33.549;
   1:L PR[91] R[100]mm/sec CNT100;
   1:  PR[GP1:91,1] = PR[GP1:90,1] + -42.479;
   1:  PR[GP1:91,2] = PR[GP1:90,2] + -34.372;
   1:L PR[91] R[100]mm/sec CNT100;
   1:  PR[GP1:91,1] = PR[GP1:90,1] + -37.583;
   1:  PR[GP1:91,2] = PR[GP1:90,2] + -34.283;
   1:L PR[91] R[100]mm/sec CNT100;
   1:  PR[GP1:91,1] = PR[GP1:90,1] + -34.567;
   1:  PR[GP1:91,2] = PR[GP1:90,2] + -33.944;
   1:L PR[91] R[100]mm/sec CNT100;
   1:  PR[GP1:91,1] = PR[GP1:90,1] + -29.773;
   1:  PR[GP1:91,2] = PR[GP1:90,2] + -32.947;
   1:L PR[91] R[100]mm/sec CNT100;
   1:  PR[GP1:91,1] = PR[GP1:90,1] + -25.247;
   1:  PR[GP1:91,2] = PR[GP1:90,2] + -31.076;
   1:L PR[91] R[100]mm/sec CNT100;
   1:  PR[GP1:91,1] = PR[GP1:90,1] + -22.565;
   1:  PR[GP1:91,2] = PR[GP1:90,2] + -29.660;
   1:L PR[91] R[100]mm/sec CNT100;
   1:  PR[GP1:91,1] = PR[GP1:90,1] + -18.466;
   1:  PR[GP1:91,2] = PR[GP1:90,2] + -26.980;
   1:L PR[91] R[100]mm/sec CNT100;
   1:  PR[GP1:91,1] = PR[GP1:90,1] + -14.936;
   1:  PR[GP1:91,2] = PR[GP1:90,2] + -23.585;
   1:L PR[91] R[100]mm/sec CNT100;
   1:  PR[GP1:91,1] = PR[GP1:90,1] + -12.955;
   1:  PR[GP1:91,2] = PR[GP1:90,2] + -21.286;
   1:L PR[91] R[100]mm/sec CNT100;
   1:  PR[GP1:91,1] = PR[GP1:90,1] + -10.118;
   1:  PR[GP1:91,2] = PR[GP1:90,2] + -17.295;
   1:L PR[91] R[100]mm/sec CNT100;
   1:  PR[GP1:91,1] = PR[GP1:90,1] + -8.072;
   1:  PR[GP1:91,2] = PR[GP1:90,2] + -12.845;
   1:L PR[91] R[100]mm/sec CNT100;
   1:  PR[GP1:91,1] = PR[GP1:90,1] + -7.068;
   1:  PR[GP1:91,2] = PR[GP1:90,2] + -9.984;
   1:L PR[91] R[100]mm/sec CNT100;
   1:  PR[GP1:91,1] = PR[GP1:90,1] + -5.853;
   1:  PR[GP1:91,2] = PR[GP1:90,2] + -5.100;
   1:L PR[91] R[100]mm/sec CNT100;
   1:  PR[GP1:91,1] = PR[GP1:90,1] + -4.023;
   1:  PR[GP1:91,2] = PR[GP1:90,2] + -1.795;
   1:L PR[91] R[100]mm/sec CNT100;
   1:  PR[GP1:91,1] = PR[GP1:90,1] + -0.454;
   1:  PR[GP1:91,2] = PR[GP1:90,2] + -0.472;
   1:L PR[91] R[100]mm/sec CNT100;
   1:  PR[GP1:91,1] = PR[GP1:90,1] + 0.667;
   1:L PR[91] R[100]mm/sec CNT100;
   1:  PR[GP1:91,1] = PR[GP1:90,1] + 4.236;
   1:  PR[GP1:91,2] = PR[GP1:90,2] + -1.795;
   1:L PR[91] R[100]mm/sec CNT100;
   1:  PR[GP1:91,1] = PR[GP1:90,1] + 6.052;
   1:  PR[GP1:91,2] = PR[GP1:90,2] + -5.076;
   1:L PR[91] R[100]mm/sec CNT100;
   1:  PR[GP1:91,1] = PR[GP1:90,1] + 7.101;
   1:  PR[GP1:91,2] = PR[GP1:90,2] + -8.064;
   1:L PR[91] R[100]mm/sec CNT100;
   1:  PR[GP1:91,1] = PR[GP1:90,1] + 8.297;
   1:  PR[GP1:91,2] = PR[GP1:90,2] + -12.871;
   1:L PR[91] R[100]mm/sec CNT100;
   1:  PR[GP1:91,1] = PR[GP1:90,1] + 10.320;
   1:  PR[GP1:91,2] = PR[GP1:90,2] + -17.269;
   1:L PR[91] R[100]mm/sec CNT100;
   1:  PR[GP1:91,1] = PR[GP1:90,1] + 12.300;
   1:  PR[GP1:91,2] = PR[GP1:90,2] + -19.567;
   1:L PR[91] R[100]mm/sec CNT100;
   1:  PR[GP1:91,1] = PR[GP1:90,1] + 15.170;
   1:  PR[GP1:91,2] = PR[GP1:90,2] + -23.605;
   1:L PR[91] R[100]mm/sec CNT100;
   1:  PR[GP1:91,1] = PR[GP1:90,1] + 18.659;
   1:  PR[GP1:91,2] = PR[GP1:90,2] + -26.960;
   1:L PR[91] R[100]mm/sec CNT100;
   1:  PR[GP1:91,1] = PR[GP1:90,1] + 21.340;
   1:  PR[GP1:91,2] = PR[GP1:90,2] + -28.376;
   1:L PR[91] R[100]mm/sec CNT100;
   1:  PR[GP1:91,1] = PR[GP1:90,1] + 25.486;
   1:  PR[GP1:91,2] = PR[GP1:90,2] + -31.086;
   1:L PR[91] R[100]mm/sec CNT100;
   1:  PR[GP1:91,1] = PR[GP1:90,1] + 29.960;
   1:  PR[GP1:91,2] = PR[GP1:90,2] + -32.936;
   1:L PR[91] R[100]mm/sec CNT100;
   1:  PR[GP1:91,1] = PR[GP1:90,1] + 32.974;
   1:  PR[GP1:91,2] = PR[GP1:90,2] + -33.274;
   1:L PR[91] R[100]mm/sec CNT100;
   1:  PR[GP1:91,1] = PR[GP1:90,1] + 37.824;
   1:  PR[GP1:91,2] = PR[GP1:90,2] + -34.283;
   1:L PR[91] R[100]mm/sec CNT100;
   1:  PR[GP1:91,1] = PR[GP1:90,1] + 42.664;
   1:  PR[GP1:91,2] = PR[GP1:90,2] + -34.371;
   1:L PR[91] R[100]mm/sec CNT100;
   1:  PR[GP1:91,1] = PR[GP1:90,1] + 45.594;
   1:  PR[GP1:91,2] = PR[GP1:90,2] + -33.585;
   1:L PR[91] R[100]mm/sec CNT100;
   1:  PR[GP1:91,1] = PR[GP1:90,1] + 50.477;
   1:  PR[GP1:91,2] = PR[GP1:90,2] + -32.754;
   1:L PR[91] R[100]mm/sec CNT100;
   1:  PR[GP1:91,1] = PR[GP1:90,1] + 55.015;
   1:  PR[GP1:91,2] = PR[GP1:90,2] + -31.068;
   1:L PR[91] R[100]mm/sec CNT100;
   1:  PR[GP1:91,1] = PR[GP1:90,1] + 57.455;
   1:  PR[GP1:91,2] = PR[GP1:90,2] + -29.267;
   1:L PR[91] R[100]mm/sec CNT100;
   1:  PR[GP1:91,1] = PR[GP1:90,1] + 61.696;
   1:  PR[GP1:91,2] = PR[GP1:90,2] + -26.709;
   1:L PR[91] R[100]mm/sec CNT100;
   1:  PR[GP1:91,1] = PR[GP1:90,1] + 65.305;
   1:  PR[GP1:91,2] = PR[GP1:90,2] + -23.482;
   1:L PR[91] R[100]mm/sec CNT100;
   1:  PR[GP1:91,1] = PR[GP1:90,1] + 66.919;
   1:  PR[GP1:91,2] = PR[GP1:90,2] + -20.913;
   1:L PR[91] R[100]mm/sec CNT100;
   1:  PR[GP1:91,1] = PR[GP1:90,1] + 69.934;
   1:  PR[GP1:91,2] = PR[GP1:90,2] + -16.982;
   1:L PR[91] R[100]mm/sec CNT100;
   1:  PR[GP1:91,1] = PR[GP1:90,1] + 72.115;
   1:  PR[GP1:91,2] = PR[GP1:90,2] + -12.661;
   1:L PR[91] R[100]mm/sec CNT100;
   1:  PR[GP1:91,1] = PR[GP1:90,1] + 72.679;
   1:  PR[GP1:91,2] = PR[GP1:90,2] + -9.680;
   1:L PR[91] R[100]mm/sec CNT100;
   1:  PR[GP1:91,1] = PR[GP1:90,1] + 74.050;
   1:  PR[GP1:91,2] = PR[GP1:90,2] + -4.920;
   1:L PR[91] R[100]mm/sec CNT100;
   1:  PR[GP1:91,1] = PR[GP1:90,1] + 74.501;
   1:  PR[GP1:91,2] = PR[GP1:90,2] + -0.100;
   1:L PR[91] R[100]mm/sec CNT100;
   1:  PR[GP1:91,1] = PR[GP1:90,1] + 73.937;
   1:  PR[GP1:91,2] = PR[GP1:90,2] + 2.880;
   1:L PR[91] R[100]mm/sec CNT100;
   1:  PR[GP1:91,1] = PR[GP1:90,1] + 73.475;
   1:  PR[GP1:91,2] = PR[GP1:90,2] + 7.812;
   1:L PR[91] R[100]mm/sec CNT100;
   1:  PR[GP1:91,1] = PR[GP1:90,1] + 72.127;
   1:  PR[GP1:91,2] = PR[GP1:90,2] + 12.491;
   1:L PR[91] R[100]mm/sec CNT100;
   1:  PR[GP1:91,1] = PR[GP1:90,1] + 69.921;
   1:  PR[GP1:91,2] = PR[GP1:90,2] + 16.863;
   1:L PR[91] R[100]mm/sec CNT100;
   1:  PR[GP1:91,1] = PR[GP1:90,1] + 68.307;
   1:  PR[GP1:91,2] = PR[GP1:90,2] + 19.433;
   1:L PR[91] R[100]mm/sec CNT100;
   1:  PR[GP1:91,1] = PR[GP1:90,1] + 65.326;
   1:  PR[GP1:91,2] = PR[GP1:90,2] + 23.319;
   1:L PR[91] R[100]mm/sec CNT100;
   1:  PR[GP1:91,1] = PR[GP1:90,1] + 61.675;
   1:  PR[GP1:91,2] = PR[GP1:90,2] + 26.584;
   1:L PR[91] R[100]mm/sec CNT100;
   1:  PR[GP1:91,1] = PR[GP1:90,1] + 59.235;
   1:  PR[GP1:91,2] = PR[GP1:90,2] + 28.385;
   1:L PR[91] R[100]mm/sec CNT100;
   1:  PR[GP1:91,1] = PR[GP1:90,1] + 55.042;
   1:  PR[GP1:91,2] = PR[GP1:90,2] + 30.914;
   1:L PR[91] R[100]mm/sec CNT100;
   1:  PR[GP1:91,1] = PR[GP1:90,1] + 50.451;
   1:  PR[GP1:91,2] = PR[GP1:90,2] + 32.619;
   1:L PR[91] R[100]mm/sec CNT100;
   1:  PR[GP1:91,1] = PR[GP1:90,1] + 47.520;
   1:  PR[GP1:91,2] = PR[GP1:90,2] + 33.405;
   1:L PR[91] R[100]mm/sec CNT100;
   1:  PR[GP1:91,1] = PR[GP1:90,1] + 42.692;
   1:  PR[GP1:91,2] = PR[GP1:90,2] + 34.228;
   1:L PR[91] R[100]mm/sec CNT100;
   1:  PR[GP1:91,1] = PR[GP1:90,1] + 37.796;
   1:  PR[GP1:91,2] = PR[GP1:90,2] + 34.139;
   1:L PR[91] R[100]mm/sec CNT100;
   1:  PR[GP1:91,1] = PR[GP1:90,1] + 34.781;
   1:  PR[GP1:91,2] = PR[GP1:90,2] + 33.800;
   1:L PR[91] R[100]mm/sec CNT100;
   1:  PR[GP1:91,1] = PR[GP1:90,1] + 29.986;
   1:  PR[GP1:91,2] = PR[GP1:90,2] + 32.803;
   1:L PR[91] R[100]mm/sec CNT100;
   1:  PR[GP1:91,1] = PR[GP1:90,1] + 25.460;
   1:  PR[GP1:91,2] = PR[GP1:90,2] + 30.932;
   1:L PR[91] R[100]mm/sec CNT100;
   1:  PR[GP1:91,1] = PR[GP1:90,1] + 22.778;
   1:  PR[GP1:91,2] = PR[GP1:90,2] + 29.516;
   1:L PR[91] R[100]mm/sec CNT100;
   1:  PR[GP1:91,1] = PR[GP1:90,1] + 18.679;
   1:  PR[GP1:91,2] = PR[GP1:90,2] + 26.836;
   1:L PR[91] R[100]mm/sec CNT100;
   1:  PR[GP1:91,1] = PR[GP1:90,1] + 15.150;
   1:  PR[GP1:91,2] = PR[GP1:90,2] + 23.441;
   1:L PR[91] R[100]mm/sec CNT100;
   1:  PR[GP1:91,1] = PR[GP1:90,1] + 13.169;
   1:  PR[GP1:91,2] = PR[GP1:90,2] + 21.142;
   1:L PR[91] R[100]mm/sec CNT100;
   1:  PR[GP1:91,1] = PR[GP1:90,1] + 10.332;
   1:  PR[GP1:91,2] = PR[GP1:90,2] + 17.151;
   1:L PR[91] R[100]mm/sec CNT100;
   1:  PR[GP1:91,1] = PR[GP1:90,1] + 8.286;
   1:  PR[GP1:91,2] = PR[GP1:90,2] + 12.701;
   1:L PR[91] R[100]mm/sec CNT100;
   1:  PR[GP1:91,1] = PR[GP1:90,1] + 7.282;
   1:  PR[GP1:91,2] = PR[GP1:90,2] + 9.840;
   1:L PR[91] R[100]mm/sec CNT100;
   1:  PR[GP1:91,1] = PR[GP1:90,1] + 6.066;
   1:  PR[GP1:91,2] = PR[GP1:90,2] + 4.956;
   1:L PR[91] R[100]mm/sec CNT100;
   1:  PR[GP1:91,1] = PR[GP1:90,1] + 4.236;
   1:  PR[GP1:91,2] = PR[GP1:90,2] + 1.651;
   1:L PR[91] R[100]mm/sec CNT100;
   1:  PR[GP1:91,1] = PR[GP1:90,1] + 0.667;
   1:  PR[GP1:91,2] = PR[GP1:90,2] + 0.328;
   1:L PR[91] R[100]mm/sec CNT100;
   1:  PR[GP1:91,1] = PR[GP1:90,1] + -0.454;
   1:L PR[91] R[100]mm/sec CNT100;
   1:  ! -- Layer/Ebene 11 -- !;
   1:  PR[91] = PR[90];
   1:  PR[GP1:91,1] = PR[GP1:90,1] + -4.023;
   1:  PR[GP1:91,2] = PR[GP1:90,2] + 1.651;
   1:  PR[GP1:91,3] = PR[GP1:90,3] + 7.015;
   1:L PR[91] R[100]mm/sec CNT100;
   1:  PR[GP1:91,1] = PR[GP1:90,1] + -5.839;
   1:  PR[GP1:91,2] = PR[GP1:90,2] + 4.932;
   1:L PR[91] R[100]mm/sec CNT100;
   1:  PR[GP1:91,1] = PR[GP1:90,1] + -6.559;
   1:  PR[GP1:91,2] = PR[GP1:90,2] + 6.984;
   1:L PR[91] R[100]mm/sec CNT100;
   1:  PR[GP1:91,1] = PR[GP1:90,1] + -7.876;
   1:  PR[GP1:91,2] = PR[GP1:90,2] + 12.274;
   1:L PR[91] R[100]mm/sec CNT100;
   1:  PR[GP1:91,1] = PR[GP1:90,1] + -10.107;
   1:  PR[GP1:91,2] = PR[GP1:90,2] + 17.125;
   1:L PR[91] R[100]mm/sec CNT100;
   1:  PR[GP1:91,1] = PR[GP1:90,1] + -11.439;
   1:  PR[GP1:91,2] = PR[GP1:90,2] + 18.672;
   1:L PR[91] R[100]mm/sec CNT100;
   1:  PR[GP1:91,1] = PR[GP1:90,1] + -14.598;
   1:  PR[GP1:91,2] = PR[GP1:90,2] + 23.115;
   1:L PR[91] R[100]mm/sec CNT100;
   1:  PR[GP1:91,1] = PR[GP1:90,1] + -18.446;
   1:  PR[GP1:91,2] = PR[GP1:90,2] + 26.816;
   1:L PR[91] R[100]mm/sec CNT100;
   1:  PR[GP1:91,1] = PR[GP1:90,1] + -20.250;
   1:  PR[GP1:91,2] = PR[GP1:90,2] + 27.769;
   1:L PR[91] R[100]mm/sec CNT100;
   1:  PR[GP1:91,1] = PR[GP1:90,1] + -24.813;
   1:  PR[GP1:91,2] = PR[GP1:90,2] + 30.752;
   1:L PR[91] R[100]mm/sec CNT100;
   1:  PR[GP1:91,1] = PR[GP1:90,1] + -29.747;
   1:  PR[GP1:91,2] = PR[GP1:90,2] + 32.792;
   1:L PR[91] R[100]mm/sec CNT100;
   1:  PR[GP1:91,1] = PR[GP1:90,1] + -31.776;
   1:  PR[GP1:91,2] = PR[GP1:90,2] + 33.020;
   1:L PR[91] R[100]mm/sec CNT100;
   1:  PR[GP1:91,1] = PR[GP1:90,1] + -37.113;
   1:  PR[GP1:91,2] = PR[GP1:90,2] + 34.130;
   1:L PR[91] R[100]mm/sec CNT100;
   1:  PR[GP1:91,1] = PR[GP1:90,1] + -42.451;
   1:  PR[GP1:91,2] = PR[GP1:90,2] + 34.227;
   1:L PR[91] R[100]mm/sec CNT100;
   1:  PR[GP1:91,1] = PR[GP1:90,1] + -44.423;
   1:  PR[GP1:91,2] = PR[GP1:90,2] + 33.699;
   1:L PR[91] R[100]mm/sec CNT100;
   1:  PR[GP1:91,1] = PR[GP1:90,1] + -49.797;
   1:  PR[GP1:91,2] = PR[GP1:90,2] + 32.783;
   1:L PR[91] R[100]mm/sec CNT100;
   1:  PR[GP1:91,1] = PR[GP1:90,1] + -54.802;
   1:  PR[GP1:91,2] = PR[GP1:90,2] + 30.924;
   1:L PR[91] R[100]mm/sec CNT100;
   1:  PR[GP1:91,1] = PR[GP1:90,1] + -56.444;
   1:  PR[GP1:91,2] = PR[GP1:90,2] + 29.712;
   1:L PR[91] R[100]mm/sec CNT100;
   1:  PR[GP1:91,1] = PR[GP1:90,1] + -61.112;
   1:  PR[GP1:91,2] = PR[GP1:90,2] + 26.896;
   1:L PR[91] R[100]mm/sec CNT100;
   1:  PR[GP1:91,1] = PR[GP1:90,1] + -65.092;
   1:  PR[GP1:91,2] = PR[GP1:90,2] + 23.338;
   1:L PR[91] R[100]mm/sec CNT100;
   1:  PR[GP1:91,1] = PR[GP1:90,1] + -66.178;
   1:  PR[GP1:91,2] = PR[GP1:90,2] + 21.609;
   1:L PR[91] R[100]mm/sec CNT100;
   1:  PR[GP1:91,1] = PR[GP1:90,1] + -69.496;
   1:  PR[GP1:91,2] = PR[GP1:90,2] + 17.283;
   1:L PR[91] R[100]mm/sec CNT100;
   1:  PR[GP1:91,1] = PR[GP1:90,1] + -71.902;
   1:  PR[GP1:91,2] = PR[GP1:90,2] + 12.516;
   1:L PR[91] R[100]mm/sec CNT100;
   1:  PR[GP1:91,1] = PR[GP1:90,1] + -72.281;
   1:  PR[GP1:91,2] = PR[GP1:90,2] + 10.511;
   1:L PR[91] R[100]mm/sec CNT100;
   1:  PR[GP1:91,1] = PR[GP1:90,1] + -73.790;
   1:  PR[GP1:91,2] = PR[GP1:90,2] + 5.272;
   1:L PR[91] R[100]mm/sec CNT100;
   1:  PR[GP1:91,1] = PR[GP1:90,1] + -74.288;
   1:  PR[GP1:91,2] = PR[GP1:90,2] + -0.044;
   1:L PR[91] R[100]mm/sec CNT100;
   1:  PR[GP1:91,1] = PR[GP1:90,1] + -73.909;
   1:  PR[GP1:91,2] = PR[GP1:90,2] + -2.050;
   1:L PR[91] R[100]mm/sec CNT100;
   1:  PR[GP1:91,1] = PR[GP1:90,1] + -73.400;
   1:  PR[GP1:91,2] = PR[GP1:90,2] + -7.477;
   1:L PR[91] R[100]mm/sec CNT100;
   1:  PR[GP1:91,1] = PR[GP1:90,1] + -71.914;
   1:  PR[GP1:91,2] = PR[GP1:90,2] + -12.635;
   1:L PR[91] R[100]mm/sec CNT100;
   1:  PR[GP1:91,1] = PR[GP1:90,1] + -69.484;
   1:  PR[GP1:91,2] = PR[GP1:90,2] + -17.452;
   1:L PR[91] R[100]mm/sec CNT100;
   1:  PR[GP1:91,1] = PR[GP1:90,1] + -68.397;
   1:  PR[GP1:91,2] = PR[GP1:90,2] + -19.182;
   1:L PR[91] R[100]mm/sec CNT100;
   1:  PR[GP1:91,1] = PR[GP1:90,1] + -65.113;
   1:  PR[GP1:91,2] = PR[GP1:90,2] + -23.463;
   1:L PR[91] R[100]mm/sec CNT100;
   1:  PR[GP1:91,1] = PR[GP1:90,1] + -61.091;
   1:  PR[GP1:91,2] = PR[GP1:90,2] + -27.059;
   1:L PR[91] R[100]mm/sec CNT100;
   1:  PR[GP1:91,1] = PR[GP1:90,1] + -59.449;
   1:  PR[GP1:91,2] = PR[GP1:90,2] + -28.272;
   1:L PR[91] R[100]mm/sec CNT100;
   1:  PR[GP1:91,1] = PR[GP1:90,1] + -54.828;
   1:  PR[GP1:91,2] = PR[GP1:90,2] + -31.058;
   1:L PR[91] R[100]mm/sec CNT100;
   1:  PR[GP1:91,1] = PR[GP1:90,1] + -49.771;
   1:  PR[GP1:91,2] = PR[GP1:90,2] + -32.937;
   1:L PR[91] R[100]mm/sec CNT100;
   1:  PR[GP1:91,1] = PR[GP1:90,1] + -47.798;
   1:  PR[GP1:91,2] = PR[GP1:90,2] + -33.466;
   1:L PR[91] R[100]mm/sec CNT100;
   1:  PR[GP1:91,1] = PR[GP1:90,1] + -42.480;
   1:  PR[GP1:91,2] = PR[GP1:90,2] + -34.372;
   1:L PR[91] R[100]mm/sec CNT100;
   1:  PR[GP1:91,1] = PR[GP1:90,1] + -37.085;
   1:  PR[GP1:91,2] = PR[GP1:90,2] + -34.274;
   1:L PR[91] R[100]mm/sec CNT100;
   1:  PR[GP1:91,1] = PR[GP1:90,1] + -35.056;
   1:  PR[GP1:91,2] = PR[GP1:90,2] + -34.046;
   1:L PR[91] R[100]mm/sec CNT100;
   1:  PR[GP1:91,1] = PR[GP1:90,1] + -29.773;
   1:  PR[GP1:91,2] = PR[GP1:90,2] + -32.947;
   1:L PR[91] R[100]mm/sec CNT100;
   1:  PR[GP1:91,1] = PR[GP1:90,1] + -24.787;
   1:  PR[GP1:91,2] = PR[GP1:90,2] + -30.885;
   1:L PR[91] R[100]mm/sec CNT100;
   1:  PR[GP1:91,1] = PR[GP1:90,1] + -22.982;
   1:  PR[GP1:91,2] = PR[GP1:90,2] + -29.932;
   1:L PR[91] R[100]mm/sec CNT100;
   1:  PR[GP1:91,1] = PR[GP1:90,1] + -18.466;
   1:  PR[GP1:91,2] = PR[GP1:90,2] + -26.980;
   1:L PR[91] R[100]mm/sec CNT100;
   1:  PR[GP1:91,1] = PR[GP1:90,1] + -14.577;
   1:  PR[GP1:91,2] = PR[GP1:90,2] + -23.240;
   1:L PR[91] R[100]mm/sec CNT100;
   1:  PR[GP1:91,1] = PR[GP1:90,1] + -13.244;
   1:  PR[GP1:91,2] = PR[GP1:90,2] + -21.693;
   1:L PR[91] R[100]mm/sec CNT100;
   1:  PR[GP1:91,1] = PR[GP1:90,1] + -10.118;
   1:  PR[GP1:91,2] = PR[GP1:90,2] + -17.295;
   1:L PR[91] R[100]mm/sec CNT100;
   1:  PR[GP1:91,1] = PR[GP1:90,1] + -7.864;
   1:  PR[GP1:91,2] = PR[GP1:90,2] + -12.393;
   1:L PR[91] R[100]mm/sec CNT100;
   1:  PR[GP1:91,1] = PR[GP1:90,1] + -7.189;
   1:  PR[GP1:91,2] = PR[GP1:90,2] + -10.467;
   1:L PR[91] R[100]mm/sec CNT100;
   1:  PR[GP1:91,1] = PR[GP1:90,1] + -5.853;
   1:  PR[GP1:91,2] = PR[GP1:90,2] + -5.100;
   1:L PR[91] R[100]mm/sec CNT100;
   1:  PR[GP1:91,1] = PR[GP1:90,1] + -4.023;
   1:  PR[GP1:91,2] = PR[GP1:90,2] + -1.795;
   1:L PR[91] R[100]mm/sec CNT100;
   1:  PR[GP1:91,1] = PR[GP1:90,1] + -0.454;
   1:  PR[GP1:91,2] = PR[GP1:90,2] + -0.472;
   1:L PR[91] R[100]mm/sec CNT100;
   1:  PR[GP1:91,1] = PR[GP1:90,1] + 0.667;
   1:L PR[91] R[100]mm/sec CNT100;
   1:  PR[GP1:91,1] = PR[GP1:90,1] + 4.236;
   1:  PR[GP1:91,2] = PR[GP1:90,2] + -1.795;
   1:L PR[91] R[100]mm/sec CNT100;
   1:  PR[GP1:91,1] = PR[GP1:90,1] + 6.052;
   1:  PR[GP1:91,2] = PR[GP1:90,2] + -5.076;
   1:L PR[91] R[100]mm/sec CNT100;
   1:  PR[GP1:91,1] = PR[GP1:90,1] + 6.772;
   1:  PR[GP1:91,2] = PR[GP1:90,2] + -7.128;
   1:L PR[91] R[100]mm/sec CNT100;
   1:  PR[GP1:91,1] = PR[GP1:90,1] + 8.090;
   1:  PR[GP1:91,2] = PR[GP1:90,2] + -12.418;
   1:L PR[91] R[100]mm/sec CNT100;
   1:  PR[GP1:91,1] = PR[GP1:90,1] + 10.320;
   1:  PR[GP1:91,2] = PR[GP1:90,2] + -17.269;
   1:L PR[91] R[100]mm/sec CNT100;
   1:  PR[GP1:91,1] = PR[GP1:90,1] + 11.653;
   1:  PR[GP1:91,2] = PR[GP1:90,2] + -18.816;
   1:L PR[91] R[100]mm/sec CNT100;
   1:  PR[GP1:91,1] = PR[GP1:90,1] + 14.811;
   1:  PR[GP1:91,2] = PR[GP1:90,2] + -23.259;
   1:L PR[91] R[100]mm/sec CNT100;
   1:  PR[GP1:91,1] = PR[GP1:90,1] + 18.659;
   1:  PR[GP1:91,2] = PR[GP1:90,2] + -26.960;
   1:L PR[91] R[100]mm/sec CNT100;
   1:  PR[GP1:91,1] = PR[GP1:90,1] + 20.463;
   1:  PR[GP1:91,2] = PR[GP1:90,2] + -27.913;
   1:L PR[91] R[100]mm/sec CNT100;
   1:  PR[GP1:91,1] = PR[GP1:90,1] + 25.026;
   1:  PR[GP1:91,2] = PR[GP1:90,2] + -30.896;
   1:L PR[91] R[100]mm/sec CNT100;
   1:  PR[GP1:91,1] = PR[GP1:90,1] + 29.960;
   1:  PR[GP1:91,2] = PR[GP1:90,2] + -32.936;
   1:L PR[91] R[100]mm/sec CNT100;
   1:  PR[GP1:91,1] = PR[GP1:90,1] + 31.989;
   1:  PR[GP1:91,2] = PR[GP1:90,2] + -33.164;
   1:L PR[91] R[100]mm/sec CNT100;
   1:  PR[GP1:91,1] = PR[GP1:90,1] + 37.326;
   1:  PR[GP1:91,2] = PR[GP1:90,2] + -34.274;
   1:L PR[91] R[100]mm/sec CNT100;
   1:  PR[GP1:91,1] = PR[GP1:90,1] + 42.664;
   1:  PR[GP1:91,2] = PR[GP1:90,2] + -34.371;
   1:L PR[91] R[100]mm/sec CNT100;
   1:  PR[GP1:91,1] = PR[GP1:90,1] + 44.636;
   1:  PR[GP1:91,2] = PR[GP1:90,2] + -33.842;
   1:L PR[91] R[100]mm/sec CNT100;
   1:  PR[GP1:91,1] = PR[GP1:90,1] + 50.010;
   1:  PR[GP1:91,2] = PR[GP1:90,2] + -32.927;
   1:L PR[91] R[100]mm/sec CNT100;
   1:  PR[GP1:91,1] = PR[GP1:90,1] + 55.015;
   1:  PR[GP1:91,2] = PR[GP1:90,2] + -31.068;
   1:L PR[91] R[100]mm/sec CNT100;
   1:  PR[GP1:91,1] = PR[GP1:90,1] + 56.657;
   1:  PR[GP1:91,2] = PR[GP1:90,2] + -29.856;
   1:L PR[91] R[100]mm/sec CNT100;
   1:  PR[GP1:91,1] = PR[GP1:90,1] + 61.325;
   1:  PR[GP1:91,2] = PR[GP1:90,2] + -27.040;
   1:L PR[91] R[100]mm/sec CNT100;
   1:  PR[GP1:91,1] = PR[GP1:90,1] + 65.305;
   1:  PR[GP1:91,2] = PR[GP1:90,2] + -23.482;
   1:L PR[91] R[100]mm/sec CNT100;
   1:  PR[GP1:91,1] = PR[GP1:90,1] + 66.392;
   1:  PR[GP1:91,2] = PR[GP1:90,2] + -21.753;
   1:L PR[91] R[100]mm/sec CNT100;
   1:  PR[GP1:91,1] = PR[GP1:90,1] + 69.710;
   1:  PR[GP1:91,2] = PR[GP1:90,2] + -17.427;
   1:L PR[91] R[100]mm/sec CNT100;
   1:  PR[GP1:91,1] = PR[GP1:90,1] + 72.115;
   1:  PR[GP1:91,2] = PR[GP1:90,2] + -12.660;
   1:L PR[91] R[100]mm/sec CNT100;
   1:  PR[GP1:91,1] = PR[GP1:90,1] + 72.494;
   1:  PR[GP1:91,2] = PR[GP1:90,2] + -10.655;
   1:L PR[91] R[100]mm/sec CNT100;
   1:  PR[GP1:91,1] = PR[GP1:90,1] + 74.003;
   1:  PR[GP1:91,2] = PR[GP1:90,2] + -5.416;
   1:L PR[91] R[100]mm/sec CNT100;
   1:  PR[GP1:91,1] = PR[GP1:90,1] + 74.501;
   1:  PR[GP1:91,2] = PR[GP1:90,2] + -0.100;
   1:L PR[91] R[100]mm/sec CNT100;
   1:  PR[GP1:91,1] = PR[GP1:90,1] + 74.122;
   1:  PR[GP1:91,2] = PR[GP1:90,2] + 1.906;
   1:L PR[91] R[100]mm/sec CNT100;
   1:  PR[GP1:91,1] = PR[GP1:90,1] + 73.613;
   1:  PR[GP1:91,2] = PR[GP1:90,2] + 7.333;
   1:L PR[91] R[100]mm/sec CNT100;
   1:  PR[GP1:91,1] = PR[GP1:90,1] + 72.128;
   1:  PR[GP1:91,2] = PR[GP1:90,2] + 12.491;
   1:L PR[91] R[100]mm/sec CNT100;
   1:  PR[GP1:91,1] = PR[GP1:90,1] + 69.697;
   1:  PR[GP1:91,2] = PR[GP1:90,2] + 17.308;
   1:L PR[91] R[100]mm/sec CNT100;
   1:  PR[GP1:91,1] = PR[GP1:90,1] + 68.610;
   1:  PR[GP1:91,2] = PR[GP1:90,2] + 19.038;
   1:L PR[91] R[100]mm/sec CNT100;
   1:  PR[GP1:91,1] = PR[GP1:90,1] + 65.327;
   1:  PR[GP1:91,2] = PR[GP1:90,2] + 23.319;
   1:L PR[91] R[100]mm/sec CNT100;
   1:  PR[GP1:91,1] = PR[GP1:90,1] + 61.304;
   1:  PR[GP1:91,2] = PR[GP1:90,2] + 26.915;
   1:L PR[91] R[100]mm/sec CNT100;
   1:  PR[GP1:91,1] = PR[GP1:90,1] + 59.662;
   1:  PR[GP1:91,2] = PR[GP1:90,2] + 28.128;
   1:L PR[91] R[100]mm/sec CNT100;
   1:  PR[GP1:91,1] = PR[GP1:90,1] + 55.042;
   1:  PR[GP1:91,2] = PR[GP1:90,2] + 30.914;
   1:L PR[91] R[100]mm/sec CNT100;
   1:  PR[GP1:91,1] = PR[GP1:90,1] + 49.984;
   1:  PR[GP1:91,2] = PR[GP1:90,2] + 32.793;
   1:L PR[91] R[100]mm/sec CNT100;
   1:  PR[GP1:91,1] = PR[GP1:90,1] + 48.012;
   1:  PR[GP1:91,2] = PR[GP1:90,2] + 33.322;
   1:L PR[91] R[100]mm/sec CNT100;
   1:  PR[GP1:91,1] = PR[GP1:90,1] + 42.693;
   1:  PR[GP1:91,2] = PR[GP1:90,2] + 34.228;
   1:L PR[91] R[100]mm/sec CNT100;
   1:  PR[GP1:91,1] = PR[GP1:90,1] + 37.298;
   1:  PR[GP1:91,2] = PR[GP1:90,2] + 34.130;
   1:L PR[91] R[100]mm/sec CNT100;
   1:  PR[GP1:91,1] = PR[GP1:90,1] + 35.269;
   1:  PR[GP1:91,2] = PR[GP1:90,2] + 33.902;
   1:L PR[91] R[100]mm/sec CNT100;
   1:  PR[GP1:91,1] = PR[GP1:90,1] + 29.987;
   1:  PR[GP1:91,2] = PR[GP1:90,2] + 32.803;
   1:L PR[91] R[100]mm/sec CNT100;
   1:  PR[GP1:91,1] = PR[GP1:90,1] + 25.001;
   1:  PR[GP1:91,2] = PR[GP1:90,2] + 30.741;
   1:L PR[91] R[100]mm/sec CNT100;
   1:  PR[GP1:91,1] = PR[GP1:90,1] + 23.195;
   1:  PR[GP1:91,2] = PR[GP1:90,2] + 29.789;
   1:L PR[91] R[100]mm/sec CNT100;
   1:  PR[GP1:91,1] = PR[GP1:90,1] + 18.679;
   1:  PR[GP1:91,2] = PR[GP1:90,2] + 26.836;
   1:L PR[91] R[100]mm/sec CNT100;
   1:  PR[GP1:91,1] = PR[GP1:90,1] + 14.791;
   1:  PR[GP1:91,2] = PR[GP1:90,2] + 23.096;
   1:L PR[91] R[100]mm/sec CNT100;
   1:  PR[GP1:91,1] = PR[GP1:90,1] + 13.458;
   1:  PR[GP1:91,2] = PR[GP1:90,2] + 21.549;
   1:L PR[91] R[100]mm/sec CNT100;
   1:  PR[GP1:91,1] = PR[GP1:90,1] + 10.332;
   1:  PR[GP1:91,2] = PR[GP1:90,2] + 17.151;
   1:L PR[91] R[100]mm/sec CNT100;
   1:  PR[GP1:91,1] = PR[GP1:90,1] + 8.078;
   1:  PR[GP1:91,2] = PR[GP1:90,2] + 12.249;
   1:L PR[91] R[100]mm/sec CNT100;
   1:  PR[GP1:91,1] = PR[GP1:90,1] + 7.402;
   1:  PR[GP1:91,2] = PR[GP1:90,2] + 10.323;
   1:L PR[91] R[100]mm/sec CNT100;
   1:  PR[GP1:91,1] = PR[GP1:90,1] + 6.066;
   1:  PR[GP1:91,2] = PR[GP1:90,2] + 4.956;
   1:L PR[91] R[100]mm/sec CNT100;
   1:  PR[GP1:91,1] = PR[GP1:90,1] + 4.236;
   1:  PR[GP1:91,2] = PR[GP1:90,2] + 1.651;
   1:L PR[91] R[100]mm/sec CNT100;
   1:  PR[GP1:91,1] = PR[GP1:90,1] + 0.667;
   1:  PR[GP1:91,2] = PR[GP1:90,2] + 0.328;
   1:L PR[91] R[100]mm/sec CNT100;
   1:  PR[GP1:91,1] = PR[GP1:90,1] + -0.454;
   1:L PR[91] R[100]mm/sec CNT100;
   1:  ! -- Layer/Ebene 12 -- !;
   1:  PR[91] = PR[90];
   1:  PR[GP1:91,1] = PR[GP1:90,1] + -4.023;
   1:  PR[GP1:91,2] = PR[GP1:90,2] + 1.651;
   1:  PR[GP1:91,3] = PR[GP1:90,3] + 7.625;
   1:L PR[91] R[100]mm/sec CNT100;
   1:  PR[GP1:91,1] = PR[GP1:90,1] + -5.839;
   1:  PR[GP1:91,2] = PR[GP1:90,2] + 4.932;
   1:L PR[91] R[100]mm/sec CNT100;
   1:  PR[GP1:91,1] = PR[GP1:90,1] + -6.231;
   1:  PR[GP1:91,2] = PR[GP1:90,2] + 6.049;
   1:L PR[91] R[100]mm/sec CNT100;
   1:  PR[GP1:91,1] = PR[GP1:90,1] + -7.668;
   1:  PR[GP1:91,2] = PR[GP1:90,2] + 11.822;
   1:L PR[91] R[100]mm/sec CNT100;
   1:  PR[GP1:91,1] = PR[GP1:90,1] + -10.107;
   1:  PR[GP1:91,2] = PR[GP1:90,2] + 17.126;
   1:L PR[91] R[100]mm/sec CNT100;
   1:  PR[GP1:91,1] = PR[GP1:90,1] + -10.792;
   1:  PR[GP1:91,2] = PR[GP1:90,2] + 17.921;
   1:L PR[91] R[100]mm/sec CNT100;
   1:  PR[GP1:91,1] = PR[GP1:90,1] + -14.239;
   1:  PR[GP1:91,2] = PR[GP1:90,2] + 22.770;
   1:L PR[91] R[100]mm/sec CNT100;
   1:  PR[GP1:91,1] = PR[GP1:90,1] + -18.446;
   1:  PR[GP1:91,2] = PR[GP1:90,2] + 26.817;
   1:L PR[91] R[100]mm/sec CNT100;
   1:  PR[GP1:91,1] = PR[GP1:90,1] + -19.373;
   1:  PR[GP1:91,2] = PR[GP1:90,2] + 27.306;
   1:L PR[91] R[100]mm/sec CNT100;
   1:  PR[GP1:91,1] = PR[GP1:90,1] + -24.353;
   1:  PR[GP1:91,2] = PR[GP1:90,2] + 30.562;
   1:L PR[91] R[100]mm/sec CNT100;
   1:  PR[GP1:91,1] = PR[GP1:90,1] + -29.748;
   1:  PR[GP1:91,2] = PR[GP1:90,2] + 32.792;
   1:L PR[91] R[100]mm/sec CNT100;
   1:  PR[GP1:91,1] = PR[GP1:90,1] + -30.790;
   1:  PR[GP1:91,2] = PR[GP1:90,2] + 32.909;
   1:L PR[91] R[100]mm/sec CNT100;
   1:  PR[GP1:91,1] = PR[GP1:90,1] + -36.615;
   1:  PR[GP1:91,2] = PR[GP1:90,2] + 34.121;
   1:L PR[91] R[100]mm/sec CNT100;
   1:  PR[GP1:91,1] = PR[GP1:90,1] + -42.452;
   1:  PR[GP1:91,2] = PR[GP1:90,2] + 34.227;
   1:L PR[91] R[100]mm/sec CNT100;
   1:  PR[GP1:91,1] = PR[GP1:90,1] + -43.465;
   1:  PR[GP1:91,2] = PR[GP1:90,2] + 33.956;
   1:L PR[91] R[100]mm/sec CNT100;
   1:  PR[GP1:91,1] = PR[GP1:90,1] + -49.330;
   1:  PR[GP1:91,2] = PR[GP1:90,2] + 32.956;
   1:L PR[91] R[100]mm/sec CNT100;
   1:  PR[GP1:91,1] = PR[GP1:90,1] + -54.802;
   1:  PR[GP1:91,2] = PR[GP1:90,2] + 30.924;
   1:L PR[91] R[100]mm/sec CNT100;
   1:  PR[GP1:91,1] = PR[GP1:90,1] + -55.646;
   1:  PR[GP1:91,2] = PR[GP1:90,2] + 30.301;
   1:L PR[91] R[100]mm/sec CNT100;
   1:  PR[GP1:91,1] = PR[GP1:90,1] + -60.741;
   1:  PR[GP1:91,2] = PR[GP1:90,2] + 27.228;
   1:L PR[91] R[100]mm/sec CNT100;
   1:  PR[GP1:91,1] = PR[GP1:90,1] + -65.092;
   1:  PR[GP1:91,2] = PR[GP1:90,2] + 23.337;
   1:L PR[91] R[100]mm/sec CNT100;
   1:  PR[GP1:91,1] = PR[GP1:90,1] + -65.651;
   1:  PR[GP1:91,2] = PR[GP1:90,2] + 22.449;
   1:L PR[91] R[100]mm/sec CNT100;
   1:  PR[GP1:91,1] = PR[GP1:90,1] + -69.272;
   1:  PR[GP1:91,2] = PR[GP1:90,2] + 17.728;
   1:L PR[91] R[100]mm/sec CNT100;
   1:  PR[GP1:91,1] = PR[GP1:90,1] + -71.902;
   1:  PR[GP1:91,2] = PR[GP1:90,2] + 12.516;
   1:L PR[91] R[100]mm/sec CNT100;
   1:  PR[GP1:91,1] = PR[GP1:90,1] + -72.097;
   1:  PR[GP1:91,2] = PR[GP1:90,2] + 11.485;
   1:L PR[91] R[100]mm/sec CNT100;
   1:  PR[GP1:91,1] = PR[GP1:90,1] + -73.743;
   1:  PR[GP1:91,2] = PR[GP1:90,2] + 5.768;
   1:L PR[91] R[100]mm/sec CNT100;
   1:  PR[GP1:91,1] = PR[GP1:90,1] + -74.288;
   1:  PR[GP1:91,2] = PR[GP1:90,2] + -0.044;
   1:L PR[91] R[100]mm/sec CNT100;
   1:  PR[GP1:91,1] = PR[GP1:90,1] + -74.093;
   1:  PR[GP1:91,2] = PR[GP1:90,2] + -1.075;
   1:L PR[91] R[100]mm/sec CNT100;
   1:  PR[GP1:91,1] = PR[GP1:90,1] + -73.538;
   1:  PR[GP1:91,2] = PR[GP1:90,2] + -6.999;
   1:L PR[91] R[100]mm/sec CNT100;
   1:  PR[GP1:91,1] = PR[GP1:90,1] + -71.914;
   1:  PR[GP1:91,2] = PR[GP1:90,2] + -12.635;
   1:L PR[91] R[100]mm/sec CNT100;
   1:  PR[GP1:91,1] = PR[GP1:90,1] + -69.259;
   1:  PR[GP1:91,2] = PR[GP1:90,2] + -17.897;
   1:L PR[91] R[100]mm/sec CNT100;
   1:  PR[GP1:91,1] = PR[GP1:90,1] + -68.700;
   1:  PR[GP1:91,2] = PR[GP1:90,2] + -18.786;
   1:L PR[91] R[100]mm/sec CNT100;
   1:  PR[GP1:91,1] = PR[GP1:90,1] + -65.114;
   1:  PR[GP1:91,2] = PR[GP1:90,2] + -23.462;
   1:L PR[91] R[100]mm/sec CNT100;
   1:  PR[GP1:91,1] = PR[GP1:90,1] + -60.720;
   1:  PR[GP1:91,2] = PR[GP1:90,2] + -27.391;
   1:L PR[91] R[100]mm/sec CNT100;
   1:  PR[GP1:91,1] = PR[GP1:90,1] + -59.876;
   1:  PR[GP1:91,2] = PR[GP1:90,2] + -28.014;
   1:L PR[91] R[100]mm/sec CNT100;
   1:  PR[GP1:91,1] = PR[GP1:90,1] + -54.829;
   1:  PR[GP1:91,2] = PR[GP1:90,2] + -31.058;
   1:L PR[91] R[100]mm/sec CNT100;
   1:  PR[GP1:91,1] = PR[GP1:90,1] + -49.304;
   1:  PR[GP1:91,2] = PR[GP1:90,2] + -33.110;
   1:L PR[91] R[100]mm/sec CNT100;
   1:  PR[GP1:91,1] = PR[GP1:90,1] + -48.290;
   1:  PR[GP1:91,2] = PR[GP1:90,2] + -33.382;
   1:L PR[91] R[100]mm/sec CNT100;
   1:  PR[GP1:91,1] = PR[GP1:90,1] + -42.480;
   1:  PR[GP1:91,2] = PR[GP1:90,2] + -34.372;
   1:L PR[91] R[100]mm/sec CNT100;
   1:  PR[GP1:91,1] = PR[GP1:90,1] + -36.587;
   1:  PR[GP1:91,2] = PR[GP1:90,2] + -34.265;
   1:L PR[91] R[100]mm/sec CNT100;
   1:  PR[GP1:91,1] = PR[GP1:90,1] + -35.544;
   1:  PR[GP1:91,2] = PR[GP1:90,2] + -34.148;
   1:L PR[91] R[100]mm/sec CNT100;
   1:  PR[GP1:91,1] = PR[GP1:90,1] + -29.774;
   1:  PR[GP1:91,2] = PR[GP1:90,2] + -32.947;
   1:L PR[91] R[100]mm/sec CNT100;
   1:  PR[GP1:91,1] = PR[GP1:90,1] + -24.327;
   1:  PR[GP1:91,2] = PR[GP1:90,2] + -30.695;
   1:L PR[91] R[100]mm/sec CNT100;
   1:  PR[GP1:91,1] = PR[GP1:90,1] + -23.399;
   1:  PR[GP1:91,2] = PR[GP1:90,2] + -30.205;
   1:L PR[91] R[100]mm/sec CNT100;
   1:  PR[GP1:91,1] = PR[GP1:90,1] + -18.466;
   1:  PR[GP1:91,2] = PR[GP1:90,2] + -26.980;
   1:L PR[91] R[100]mm/sec CNT100;
   1:  PR[GP1:91,1] = PR[GP1:90,1] + -14.219;
   1:  PR[GP1:91,2] = PR[GP1:90,2] + -22.895;
   1:L PR[91] R[100]mm/sec CNT100;
   1:  PR[GP1:91,1] = PR[GP1:90,1] + -13.533;
   1:  PR[GP1:91,2] = PR[GP1:90,2] + -22.099;
   1:L PR[91] R[100]mm/sec CNT100;
   1:  PR[GP1:91,1] = PR[GP1:90,1] + -10.119;
   1:  PR[GP1:91,2] = PR[GP1:90,2] + -17.295;
   1:L PR[91] R[100]mm/sec CNT100;
   1:  PR[GP1:91,1] = PR[GP1:90,1] + -7.657;
   1:  PR[GP1:91,2] = PR[GP1:90,2] + -11.941;
   1:L PR[91] R[100]mm/sec CNT100;
   1:  PR[GP1:91,1] = PR[GP1:90,1] + -7.309;
   1:  PR[GP1:91,2] = PR[GP1:90,2] + -10.951;
   1:L PR[91] R[100]mm/sec CNT100;
   1:  PR[GP1:91,1] = PR[GP1:90,1] + -5.853;
   1:  PR[GP1:91,2] = PR[GP1:90,2] + -5.100;
   1:L PR[91] R[100]mm/sec CNT100;
   1:  PR[GP1:91,1] = PR[GP1:90,1] + -4.023;
   1:  PR[GP1:91,2] = PR[GP1:90,2] + -1.795;
   1:L PR[91] R[100]mm/sec CNT100;
   1:  PR[GP1:91,1] = PR[GP1:90,1] + -0.454;
   1:  PR[GP1:91,2] = PR[GP1:90,2] + -0.472;
   1:L PR[91] R[100]mm/sec CNT100;
   1:  PR[GP1:91,1] = PR[GP1:90,1] + 0.667;
   1:L PR[91] R[100]mm/sec CNT100;
   1:  PR[GP1:91,1] = PR[GP1:90,1] + 4.236;
   1:  PR[GP1:91,2] = PR[GP1:90,2] + -1.795;
   1:L PR[91] R[100]mm/sec CNT100;
   1:  PR[GP1:91,1] = PR[GP1:90,1] + 6.052;
   1:  PR[GP1:91,2] = PR[GP1:90,2] + -5.076;
   1:L PR[91] R[100]mm/sec CNT100;
   1:  PR[GP1:91,1] = PR[GP1:90,1] + 6.444;
   1:  PR[GP1:91,2] = PR[GP1:90,2] + -6.193;
   1:L PR[91] R[100]mm/sec CNT100;
   1:  PR[GP1:91,1] = PR[GP1:90,1] + 7.882;
   1:  PR[GP1:91,2] = PR[GP1:90,2] + -11.966;
   1:L PR[91] R[100]mm/sec CNT100;
   1:  PR[GP1:91,1] = PR[GP1:90,1] + 10.320;
   1:  PR[GP1:91,2] = PR[GP1:90,2] + -17.270;
   1:L PR[91] R[100]mm/sec CNT100;
   1:  PR[GP1:91,1] = PR[GP1:90,1] + 11.005;
   1:  PR[GP1:91,2] = PR[GP1:90,2] + -18.065;
   1:L PR[91] R[100]mm/sec CNT100;
   1:  PR[GP1:91,1] = PR[GP1:90,1] + 14.452;
   1:  PR[GP1:91,2] = PR[GP1:90,2] + -22.914;
   1:L PR[91] R[100]mm/sec CNT100;
   1:  PR[GP1:91,1] = PR[GP1:90,1] + 18.659;
   1:  PR[GP1:91,2] = PR[GP1:90,2] + -26.961;
   1:L PR[91] R[100]mm/sec CNT100;
   1:  PR[GP1:91,1] = PR[GP1:90,1] + 19.587;
   1:  PR[GP1:91,2] = PR[GP1:90,2] + -27.450;
   1:L PR[91] R[100]mm/sec CNT100;
   1:  PR[GP1:91,1] = PR[GP1:90,1] + 24.567;
   1:  PR[GP1:91,2] = PR[GP1:90,2] + -30.706;
   1:L PR[91] R[100]mm/sec CNT100;
   1:  PR[GP1:91,1] = PR[GP1:90,1] + 29.961;
   1:  PR[GP1:91,2] = PR[GP1:90,2] + -32.936;
   1:L PR[91] R[100]mm/sec CNT100;
   1:  PR[GP1:91,1] = PR[GP1:90,1] + 31.004;
   1:  PR[GP1:91,2] = PR[GP1:90,2] + -33.053;
   1:L PR[91] R[100]mm/sec CNT100;
   1:  PR[GP1:91,1] = PR[GP1:90,1] + 36.829;
   1:  PR[GP1:91,2] = PR[GP1:90,2] + -34.265;
   1:L PR[91] R[100]mm/sec CNT100;
   1:  PR[GP1:91,1] = PR[GP1:90,1] + 42.665;
   1:  PR[GP1:91,2] = PR[GP1:90,2] + -34.371;
   1:L PR[91] R[100]mm/sec CNT100;
   1:  PR[GP1:91,1] = PR[GP1:90,1] + 43.678;
   1:  PR[GP1:91,2] = PR[GP1:90,2] + -34.100;
   1:L PR[91] R[100]mm/sec CNT100;
   1:  PR[GP1:91,1] = PR[GP1:90,1] + 49.544;
   1:  PR[GP1:91,2] = PR[GP1:90,2] + -33.100;
   1:L PR[91] R[100]mm/sec CNT100;
   1:  PR[GP1:91,1] = PR[GP1:90,1] + 55.015;
   1:  PR[GP1:91,2] = PR[GP1:90,2] + -31.068;
   1:L PR[91] R[100]mm/sec CNT100;
   1:  PR[GP1:91,1] = PR[GP1:90,1] + 55.859;
   1:  PR[GP1:91,2] = PR[GP1:90,2] + -30.445;
   1:L PR[91] R[100]mm/sec CNT100;
   1:  PR[GP1:91,1] = PR[GP1:90,1] + 60.954;
   1:  PR[GP1:91,2] = PR[GP1:90,2] + -27.372;
   1:L PR[91] R[100]mm/sec CNT100;
   1:  PR[GP1:91,1] = PR[GP1:90,1] + 65.306;
   1:  PR[GP1:91,2] = PR[GP1:90,2] + -23.481;
   1:L PR[91] R[100]mm/sec CNT100;
   1:  PR[GP1:91,1] = PR[GP1:90,1] + 65.864;
   1:  PR[GP1:91,2] = PR[GP1:90,2] + -22.593;
   1:L PR[91] R[100]mm/sec CNT100;
   1:  PR[GP1:91,1] = PR[GP1:90,1] + 69.485;
   1:  PR[GP1:91,2] = PR[GP1:90,2] + -17.871;
   1:L PR[91] R[100]mm/sec CNT100;
   1:  PR[GP1:91,1] = PR[GP1:90,1] + 72.115;
   1:  PR[GP1:91,2] = PR[GP1:90,2] + -12.660;
   1:L PR[91] R[100]mm/sec CNT100;
   1:  PR[GP1:91,1] = PR[GP1:90,1] + 72.310;
   1:  PR[GP1:91,2] = PR[GP1:90,2] + -11.629;
   1:L PR[91] R[100]mm/sec CNT100;
   1:  PR[GP1:91,1] = PR[GP1:90,1] + 73.957;
   1:  PR[GP1:91,2] = PR[GP1:90,2] + -5.912;
   1:L PR[91] R[100]mm/sec CNT100;
   1:  PR[GP1:91,1] = PR[GP1:90,1] + 74.501;
   1:  PR[GP1:91,2] = PR[GP1:90,2] + -0.100;
   1:L PR[91] R[100]mm/sec CNT100;
   1:  PR[GP1:91,1] = PR[GP1:90,1] + 74.306;
   1:  PR[GP1:91,2] = PR[GP1:90,2] + 0.931;
   1:L PR[91] R[100]mm/sec CNT100;
   1:  PR[GP1:91,1] = PR[GP1:90,1] + 73.751;
   1:  PR[GP1:91,2] = PR[GP1:90,2] + 6.855;
   1:L PR[91] R[100]mm/sec CNT100;
   1:  PR[GP1:91,1] = PR[GP1:90,1] + 72.128;
   1:  PR[GP1:91,2] = PR[GP1:90,2] + 12.491;
   1:L PR[91] R[100]mm/sec CNT100;
   1:  PR[GP1:91,1] = PR[GP1:90,1] + 69.472;
   1:  PR[GP1:91,2] = PR[GP1:90,2] + 17.753;
   1:L PR[91] R[100]mm/sec CNT100;
   1:  PR[GP1:91,1] = PR[GP1:90,1] + 68.914;
   1:  PR[GP1:91,2] = PR[GP1:90,2] + 18.642;
   1:L PR[91] R[100]mm/sec CNT100;
   1:  PR[GP1:91,1] = PR[GP1:90,1] + 65.327;
   1:  PR[GP1:91,2] = PR[GP1:90,2] + 23.318;
   1:L PR[91] R[100]mm/sec CNT100;
   1:  PR[GP1:91,1] = PR[GP1:90,1] + 60.933;
   1:  PR[GP1:91,2] = PR[GP1:90,2] + 27.247;
   1:L PR[91] R[100]mm/sec CNT100;
   1:  PR[GP1:91,1] = PR[GP1:90,1] + 60.089;
   1:  PR[GP1:91,2] = PR[GP1:90,2] + 27.870;
   1:L PR[91] R[100]mm/sec CNT100;
   1:  PR[GP1:91,1] = PR[GP1:90,1] + 55.042;
   1:  PR[GP1:91,2] = PR[GP1:90,2] + 30.914;
   1:L PR[91] R[100]mm/sec CNT100;
   1:  PR[GP1:91,1] = PR[GP1:90,1] + 49.517;
   1:  PR[GP1:91,2] = PR[GP1:90,2] + 32.966;
   1:L PR[91] R[100]mm/sec CNT100;
   1:  PR[GP1:91,1] = PR[GP1:90,1] + 48.503;
   1:  PR[GP1:91,2] = PR[GP1:90,2] + 33.238;
   1:L PR[91] R[100]mm/sec CNT100;
   1:  PR[GP1:91,1] = PR[GP1:90,1] + 42.693;
   1:  PR[GP1:91,2] = PR[GP1:90,2] + 34.228;
   1:L PR[91] R[100]mm/sec CNT100;
   1:  PR[GP1:91,1] = PR[GP1:90,1] + 36.801;
   1:  PR[GP1:91,2] = PR[GP1:90,2] + 34.121;
   1:L PR[91] R[100]mm/sec CNT100;
   1:  PR[GP1:91,1] = PR[GP1:90,1] + 35.757;
   1:  PR[GP1:91,2] = PR[GP1:90,2] + 34.004;
   1:L PR[91] R[100]mm/sec CNT100;
   1:  PR[GP1:91,1] = PR[GP1:90,1] + 29.987;
   1:  PR[GP1:91,2] = PR[GP1:90,2] + 32.803;
   1:L PR[91] R[100]mm/sec CNT100;
   1:  PR[GP1:91,1] = PR[GP1:90,1] + 24.541;
   1:  PR[GP1:91,2] = PR[GP1:90,2] + 30.551;
   1:L PR[91] R[100]mm/sec CNT100;
   1:  PR[GP1:91,1] = PR[GP1:90,1] + 23.613;
   1:  PR[GP1:91,2] = PR[GP1:90,2] + 30.061;
   1:L PR[91] R[100]mm/sec CNT100;
   1:  PR[GP1:91,1] = PR[GP1:90,1] + 18.679;
   1:  PR[GP1:91,2] = PR[GP1:90,2] + 26.836;
   1:L PR[91] R[100]mm/sec CNT100;
   1:  PR[GP1:91,1] = PR[GP1:90,1] + 14.432;
   1:  PR[GP1:91,2] = PR[GP1:90,2] + 22.751;
   1:L PR[91] R[100]mm/sec CNT100;
   1:  PR[GP1:91,1] = PR[GP1:90,1] + 13.746;
   1:  PR[GP1:91,2] = PR[GP1:90,2] + 21.955;
   1:L PR[91] R[100]mm/sec CNT100;
   1:  PR[GP1:91,1] = PR[GP1:90,1] + 10.332;
   1:  PR[GP1:91,2] = PR[GP1:90,2] + 17.151;
   1:L PR[91] R[100]mm/sec CNT100;
   1:  PR[GP1:91,1] = PR[GP1:90,1] + 7.870;
   1:  PR[GP1:91,2] = PR[GP1:90,2] + 11.797;
   1:L PR[91] R[100]mm/sec CNT100;
   1:  PR[GP1:91,1] = PR[GP1:90,1] + 7.522;
   1:  PR[GP1:91,2] = PR[GP1:90,2] + 10.807;
   1:L PR[91] R[100]mm/sec CNT100;
   1:  PR[GP1:91,1] = PR[GP1:90,1] + 6.066;
   1:  PR[GP1:91,2] = PR[GP1:90,2] + 4.956;
   1:L PR[91] R[100]mm/sec CNT100;
   1:  PR[GP1:91,1] = PR[GP1:90,1] + 4.236;
   1:  PR[GP1:91,2] = PR[GP1:90,2] + 1.651;
   1:L PR[91] R[100]mm/sec CNT100;
   1:  PR[GP1:91,1] = PR[GP1:90,1] + 0.667;
   1:  PR[GP1:91,2] = PR[GP1:90,2] + 0.328;
   1:L PR[91] R[100]mm/sec CNT100;
   1:  PR[GP1:91,1] = PR[GP1:90,1] + -0.454;
   1:L PR[91] R[100]mm/sec CNT100;
   1:  ! -- Layer/Ebene 13 -- !;
   1:  PR[91] = PR[90];
   1:  PR[GP1:91,1] = PR[GP1:90,1] + -4.023;
   1:  PR[GP1:91,2] = PR[GP1:90,2] + 1.651;
   1:  PR[GP1:91,3] = PR[GP1:90,3] + 8.235;
   1:L PR[91] R[100]mm/sec CNT100;
   1:  PR[GP1:91,1] = PR[GP1:90,1] + -5.839;
   1:  PR[GP1:91,2] = PR[GP1:90,2] + 4.932;
   1:L PR[91] R[100]mm/sec CNT100;
   1:  PR[GP1:91,1] = PR[GP1:90,1] + -5.902;
   1:  PR[GP1:91,2] = PR[GP1:90,2] + 5.113;
   1:L PR[91] R[100]mm/sec CNT100;
   1:  PR[GP1:91,1] = PR[GP1:90,1] + -7.460;
   1:  PR[GP1:91,2] = PR[GP1:90,2] + 11.370;
   1:L PR[91] R[100]mm/sec CNT100;
   1:  PR[GP1:91,1] = PR[GP1:90,1] + -10.107;
   1:  PR[GP1:91,2] = PR[GP1:90,2] + 17.126;
   1:L PR[91] R[100]mm/sec CNT100;
   1:  PR[GP1:91,1] = PR[GP1:90,1] + -10.144;
   1:  PR[GP1:91,2] = PR[GP1:90,2] + 17.169;
   1:L PR[91] R[100]mm/sec CNT100;
   1:  PR[GP1:91,1] = PR[GP1:90,1] + -13.880;
   1:  PR[GP1:91,2] = PR[GP1:90,2] + 22.425;
   1:L PR[91] R[100]mm/sec CNT100;
   1:  PR[GP1:91,1] = PR[GP1:90,1] + -18.446;
   1:  PR[GP1:91,2] = PR[GP1:90,2] + 26.817;
   1:L PR[91] R[100]mm/sec CNT100;
   1:  PR[GP1:91,1] = PR[GP1:90,1] + -18.497;
   1:  PR[GP1:91,2] = PR[GP1:90,2] + 26.844;
   1:L PR[91] R[100]mm/sec CNT100;
   1:  PR[GP1:91,1] = PR[GP1:90,1] + -23.894;
   1:  PR[GP1:91,2] = PR[GP1:90,2] + 30.372;
   1:L PR[91] R[100]mm/sec CNT100;
   1:  PR[GP1:91,1] = PR[GP1:90,1] + -29.748;
   1:  PR[GP1:91,2] = PR[GP1:90,2] + 32.792;
   1:L PR[91] R[100]mm/sec CNT100;
   1:  PR[GP1:91,1] = PR[GP1:90,1] + -29.805;
   1:  PR[GP1:91,2] = PR[GP1:90,2] + 32.799;
   1:L PR[91] R[100]mm/sec CNT100;
   1:  PR[GP1:91,1] = PR[GP1:90,1] + -36.118;
   1:  PR[GP1:91,2] = PR[GP1:90,2] + 34.112;
   1:L PR[91] R[100]mm/sec CNT100;
   1:  PR[GP1:91,1] = PR[GP1:90,1] + -42.452;
   1:  PR[GP1:91,2] = PR[GP1:90,2] + 34.227;
   1:L PR[91] R[100]mm/sec CNT100;
   1:  PR[GP1:91,1] = PR[GP1:90,1] + -42.507;
   1:  PR[GP1:91,2] = PR[GP1:90,2] + 34.213;
   1:L PR[91] R[100]mm/sec CNT100;
   1:  PR[GP1:91,1] = PR[GP1:90,1] + -48.864;
   1:  PR[GP1:91,2] = PR[GP1:90,2] + 33.130;
   1:L PR[91] R[100]mm/sec CNT100;
   1:  PR[GP1:91,1] = PR[GP1:90,1] + -54.802;
   1:  PR[GP1:91,2] = PR[GP1:90,2] + 30.923;
   1:L PR[91] R[100]mm/sec CNT100;
   1:  PR[GP1:91,1] = PR[GP1:90,1] + -54.848;
   1:  PR[GP1:91,2] = PR[GP1:90,2] + 30.889;
   1:L PR[91] R[100]mm/sec CNT100;
   1:  PR[GP1:91,1] = PR[GP1:90,1] + -60.370;
   1:  PR[GP1:91,2] = PR[GP1:90,2] + 27.560;
   1:L PR[91] R[100]mm/sec CNT100;
   1:  PR[GP1:91,1] = PR[GP1:90,1] + -65.093;
   1:  PR[GP1:91,2] = PR[GP1:90,2] + 23.337;
   1:L PR[91] R[100]mm/sec CNT100;
   1:  PR[GP1:91,1] = PR[GP1:90,1] + -65.123;
   1:  PR[GP1:91,2] = PR[GP1:90,2] + 23.289;
   1:L PR[91] R[100]mm/sec CNT100;
   1:  PR[GP1:91,1] = PR[GP1:90,1] + -69.047;
   1:  PR[GP1:91,2] = PR[GP1:90,2] + 18.172;
   1:L PR[91] R[100]mm/sec CNT100;
   1:  PR[GP1:91,1] = PR[GP1:90,1] + -71.902;
   1:  PR[GP1:91,2] = PR[GP1:90,2] + 12.516;
   1:L PR[91] R[100]mm/sec CNT100;
   1:  PR[GP1:91,1] = PR[GP1:90,1] + -71.912;
   1:  PR[GP1:91,2] = PR[GP1:90,2] + 12.460;
   1:L PR[91] R[100]mm/sec CNT100;
   1:  PR[GP1:91,1] = PR[GP1:90,1] + -73.697;
   1:  PR[GP1:91,2] = PR[GP1:90,2] + 6.264;
   1:L PR[91] R[100]mm/sec CNT100;
   1:  PR[GP1:91,1] = PR[GP1:90,1] + -74.288;
   1:  PR[GP1:91,2] = PR[GP1:90,2] + -0.044;
   1:L PR[91] R[100]mm/sec CNT100;
   1:  PR[GP1:91,1] = PR[GP1:90,1] + -74.277;
   1:  PR[GP1:91,2] = PR[GP1:90,2] + -0.100;
   1:L PR[91] R[100]mm/sec CNT100;
   1:  PR[GP1:91,1] = PR[GP1:90,1] + -73.676;
   1:  PR[GP1:91,2] = PR[GP1:90,2] + -6.520;
   1:L PR[91] R[100]mm/sec CNT100;
   1:  PR[GP1:91,1] = PR[GP1:90,1] + -71.914;
   1:  PR[GP1:91,2] = PR[GP1:90,2] + -12.635;
   1:L PR[91] R[100]mm/sec CNT100;
   1:  PR[GP1:91,1] = PR[GP1:90,1] + -69.035;
   1:  PR[GP1:91,2] = PR[GP1:90,2] + -18.341;
   1:L PR[91] R[100]mm/sec CNT100;
   1:  PR[GP1:91,1] = PR[GP1:90,1] + -69.004;
   1:  PR[GP1:91,2] = PR[GP1:90,2] + -18.390;
   1:L PR[91] R[100]mm/sec CNT100;
   1:  PR[GP1:91,1] = PR[GP1:90,1] + -65.114;
   1:  PR[GP1:91,2] = PR[GP1:90,2] + -23.462;
   1:L PR[91] R[100]mm/sec CNT100;
   1:  PR[GP1:91,1] = PR[GP1:90,1] + -60.349;
   1:  PR[GP1:91,2] = PR[GP1:90,2] + -27.723;
   1:L PR[91] R[100]mm/sec CNT100;
   1:  PR[GP1:91,1] = PR[GP1:90,1] + -60.303;
   1:  PR[GP1:91,2] = PR[GP1:90,2] + -27.757;
   1:L PR[91] R[100]mm/sec CNT100;
   1:  PR[GP1:91,1] = PR[GP1:90,1] + -54.829;
   1:  PR[GP1:91,2] = PR[GP1:90,2] + -31.058;
   1:L PR[91] R[100]mm/sec CNT100;
   1:  PR[GP1:91,1] = PR[GP1:90,1] + -48.837;
   1:  PR[GP1:91,2] = PR[GP1:90,2] + -33.283;
   1:L PR[91] R[100]mm/sec CNT100;
   1:  PR[GP1:91,1] = PR[GP1:90,1] + -48.782;
   1:  PR[GP1:91,2] = PR[GP1:90,2] + -33.298;
   1:L PR[91] R[100]mm/sec CNT100;
   1:  PR[GP1:91,1] = PR[GP1:90,1] + -42.480;
   1:  PR[GP1:91,2] = PR[GP1:90,2] + -34.372;
   1:L PR[91] R[100]mm/sec CNT100;
   1:  PR[GP1:91,1] = PR[GP1:90,1] + -36.090;
   1:  PR[GP1:91,2] = PR[GP1:90,2] + -34.256;
   1:L PR[91] R[100]mm/sec CNT100;
   1:  PR[GP1:91,1] = PR[GP1:90,1] + -36.032;
   1:  PR[GP1:91,2] = PR[GP1:90,2] + -34.249;
   1:L PR[91] R[100]mm/sec CNT100;
   1:  PR[GP1:91,1] = PR[GP1:90,1] + -29.774;
   1:  PR[GP1:91,2] = PR[GP1:90,2] + -32.947;
   1:L PR[91] R[100]mm/sec CNT100;
   1:  PR[GP1:91,1] = PR[GP1:90,1] + -23.868;
   1:  PR[GP1:91,2] = PR[GP1:90,2] + -30.505;
   1:L PR[91] R[100]mm/sec CNT100;
   1:  PR[GP1:91,1] = PR[GP1:90,1] + -23.817;
   1:  PR[GP1:91,2] = PR[GP1:90,2] + -30.478;
   1:L PR[91] R[100]mm/sec CNT100;
   1:  PR[GP1:91,1] = PR[GP1:90,1] + -18.466;
   1:  PR[GP1:91,2] = PR[GP1:90,2] + -26.980;
   1:L PR[91] R[100]mm/sec CNT100;
   1:  PR[GP1:91,1] = PR[GP1:90,1] + -13.860;
   1:  PR[GP1:91,2] = PR[GP1:90,2] + -22.550;
   1:L PR[91] R[100]mm/sec CNT100;
   1:  PR[GP1:91,1] = PR[GP1:90,1] + -13.822;
   1:  PR[GP1:91,2] = PR[GP1:90,2] + -22.506;
   1:L PR[91] R[100]mm/sec CNT100;
   1:  PR[GP1:91,1] = PR[GP1:90,1] + -10.119;
   1:  PR[GP1:91,2] = PR[GP1:90,2] + -17.296;
   1:L PR[91] R[100]mm/sec CNT100;
   1:  PR[GP1:91,1] = PR[GP1:90,1] + -7.449;
   1:  PR[GP1:91,2] = PR[GP1:90,2] + -11.488;
   1:L PR[91] R[100]mm/sec CNT100;
   1:  PR[GP1:91,1] = PR[GP1:90,1] + -7.430;
   1:  PR[GP1:91,2] = PR[GP1:90,2] + -11.434;
   1:L PR[91] R[100]mm/sec CNT100;
   1:  PR[GP1:91,1] = PR[GP1:90,1] + -5.853;
   1:  PR[GP1:91,2] = PR[GP1:90,2] + -5.100;
   1:L PR[91] R[100]mm/sec CNT100;
   1:  PR[GP1:91,1] = PR[GP1:90,1] + -4.023;
   1:  PR[GP1:91,2] = PR[GP1:90,2] + -1.795;
   1:L PR[91] R[100]mm/sec CNT100;
   1:  PR[GP1:91,1] = PR[GP1:90,1] + -0.454;
   1:  PR[GP1:91,2] = PR[GP1:90,2] + -0.472;
   1:L PR[91] R[100]mm/sec CNT100;
   1:  PR[GP1:91,1] = PR[GP1:90,1] + 0.667;
   1:L PR[91] R[100]mm/sec CNT100;
   1:  PR[GP1:91,1] = PR[GP1:90,1] + 4.236;
   1:  PR[GP1:91,2] = PR[GP1:90,2] + -1.795;
   1:L PR[91] R[100]mm/sec CNT100;
   1:  PR[GP1:91,1] = PR[GP1:90,1] + 6.052;
   1:  PR[GP1:91,2] = PR[GP1:90,2] + -5.076;
   1:L PR[91] R[100]mm/sec CNT100;
   1:  PR[GP1:91,1] = PR[GP1:90,1] + 6.116;
   1:  PR[GP1:91,2] = PR[GP1:90,2] + -5.257;
   1:L PR[91] R[100]mm/sec CNT100;
   1:  PR[GP1:91,1] = PR[GP1:90,1] + 7.674;
   1:  PR[GP1:91,2] = PR[GP1:90,2] + -11.514;
   1:L PR[91] R[100]mm/sec CNT100;
   1:  PR[GP1:91,1] = PR[GP1:90,1] + 10.320;
   1:  PR[GP1:91,2] = PR[GP1:90,2] + -17.270;
   1:L PR[91] R[100]mm/sec CNT100;
   1:  PR[GP1:91,1] = PR[GP1:90,1] + 10.358;
   1:  PR[GP1:91,2] = PR[GP1:90,2] + -17.313;
   1:L PR[91] R[100]mm/sec CNT100;
   1:  PR[GP1:91,1] = PR[GP1:90,1] + 14.093;
   1:  PR[GP1:91,2] = PR[GP1:90,2] + -22.569;
   1:L PR[91] R[100]mm/sec CNT100;
   1:  PR[GP1:91,1] = PR[GP1:90,1] + 18.659;
   1:  PR[GP1:91,2] = PR[GP1:90,2] + -26.961;
   1:L PR[91] R[100]mm/sec CNT100;
   1:  PR[GP1:91,1] = PR[GP1:90,1] + 18.710;
   1:  PR[GP1:91,2] = PR[GP1:90,2] + -26.988;
   1:L PR[91] R[100]mm/sec CNT100;
   1:  PR[GP1:91,1] = PR[GP1:90,1] + 24.107;
   1:  PR[GP1:91,2] = PR[GP1:90,2] + -30.516;
   1:L PR[91] R[100]mm/sec CNT100;
   1:  PR[GP1:91,1] = PR[GP1:90,1] + 29.961;
   1:  PR[GP1:91,2] = PR[GP1:90,2] + -32.936;
   1:L PR[91] R[100]mm/sec CNT100;
   1:  PR[GP1:91,1] = PR[GP1:90,1] + 30.018;
   1:  PR[GP1:91,2] = PR[GP1:90,2] + -32.943;
   1:L PR[91] R[100]mm/sec CNT100;
   1:  PR[GP1:91,1] = PR[GP1:90,1] + 36.331;
   1:  PR[GP1:91,2] = PR[GP1:90,2] + -34.256;
   1:L PR[91] R[100]mm/sec CNT100;
   1:  PR[GP1:91,1] = PR[GP1:90,1] + 42.665;
   1:  PR[GP1:91,2] = PR[GP1:90,2] + -34.371;
   1:L PR[91] R[100]mm/sec CNT100;
   1:  PR[GP1:91,1] = PR[GP1:90,1] + 42.721;
   1:  PR[GP1:91,2] = PR[GP1:90,2] + -34.357;
   1:L PR[91] R[100]mm/sec CNT100;
   1:  PR[GP1:91,1] = PR[GP1:90,1] + 49.077;
   1:  PR[GP1:91,2] = PR[GP1:90,2] + -33.274;
   1:L PR[91] R[100]mm/sec CNT100;
   1:  PR[GP1:91,1] = PR[GP1:90,1] + 55.016;
   1:  PR[GP1:91,2] = PR[GP1:90,2] + -31.067;
   1:L PR[91] R[100]mm/sec CNT100;
   1:  PR[GP1:91,1] = PR[GP1:90,1] + 55.062;
   1:  PR[GP1:91,2] = PR[GP1:90,2] + -31.033;
   1:L PR[91] R[100]mm/sec CNT100;
   1:  PR[GP1:91,1] = PR[GP1:90,1] + 60.583;
   1:  PR[GP1:91,2] = PR[GP1:90,2] + -27.704;
   1:L PR[91] R[100]mm/sec CNT100;
   1:  PR[GP1:91,1] = PR[GP1:90,1] + 65.306;
   1:  PR[GP1:91,2] = PR[GP1:90,2] + -23.481;
   1:L PR[91] R[100]mm/sec CNT100;
   1:  PR[GP1:91,1] = PR[GP1:90,1] + 65.337;
   1:  PR[GP1:91,2] = PR[GP1:90,2] + -23.432;
   1:L PR[91] R[100]mm/sec CNT100;
   1:  PR[GP1:91,1] = PR[GP1:90,1] + 69.261;
   1:  PR[GP1:91,2] = PR[GP1:90,2] + -18.316;
   1:L PR[91] R[100]mm/sec CNT100;
   1:  PR[GP1:91,1] = PR[GP1:90,1] + 72.115;
   1:  PR[GP1:91,2] = PR[GP1:90,2] + -12.660;
   1:L PR[91] R[100]mm/sec CNT100;
   1:  PR[GP1:91,1] = PR[GP1:90,1] + 72.126;
   1:  PR[GP1:91,2] = PR[GP1:90,2] + -12.604;
   1:L PR[91] R[100]mm/sec CNT100;
   1:  PR[GP1:91,1] = PR[GP1:90,1] + 73.910;
   1:  PR[GP1:91,2] = PR[GP1:90,2] + -6.408;
   1:L PR[91] R[100]mm/sec CNT100;
   1:  PR[GP1:91,1] = PR[GP1:90,1] + 74.501;
   1:  PR[GP1:91,2] = PR[GP1:90,2] + -0.100;
   1:L PR[91] R[100]mm/sec CNT100;
   1:  PR[GP1:91,1] = PR[GP1:90,1] + 74.491;
   1:  PR[GP1:91,2] = PR[GP1:90,2] + -0.044;
   1:L PR[91] R[100]mm/sec CNT100;
   1:  PR[GP1:91,1] = PR[GP1:90,1] + 73.889;
   1:  PR[GP1:91,2] = PR[GP1:90,2] + 6.376;
   1:L PR[91] R[100]mm/sec CNT100;
   1:  PR[GP1:91,1] = PR[GP1:90,1] + 72.128;
   1:  PR[GP1:91,2] = PR[GP1:90,2] + 12.491;
   1:L PR[91] R[100]mm/sec CNT100;
   1:  PR[GP1:91,1] = PR[GP1:90,1] + 69.248;
   1:  PR[GP1:91,2] = PR[GP1:90,2] + 18.197;
   1:L PR[91] R[100]mm/sec CNT100;
   1:  PR[GP1:91,1] = PR[GP1:90,1] + 69.217;
   1:  PR[GP1:91,2] = PR[GP1:90,2] + 18.246;
   1:L PR[91] R[100]mm/sec CNT100;
   1:  PR[GP1:91,1] = PR[GP1:90,1] + 65.327;
   1:  PR[GP1:91,2] = PR[GP1:90,2] + 23.318;
   1:L PR[91] R[100]mm/sec CNT100;
   1:  PR[GP1:91,1] = PR[GP1:90,1] + 60.562;
   1:  PR[GP1:91,2] = PR[GP1:90,2] + 27.579;
   1:L PR[91] R[100]mm/sec CNT100;
   1:  PR[GP1:91,1] = PR[GP1:90,1] + 60.516;
   1:  PR[GP1:91,2] = PR[GP1:90,2] + 27.613;
   1:L PR[91] R[100]mm/sec CNT100;
   1:  PR[GP1:91,1] = PR[GP1:90,1] + 55.042;
   1:  PR[GP1:91,2] = PR[GP1:90,2] + 30.914;
   1:L PR[91] R[100]mm/sec CNT100;
   1:  PR[GP1:91,1] = PR[GP1:90,1] + 49.051;
   1:  PR[GP1:91,2] = PR[GP1:90,2] + 33.139;
   1:L PR[91] R[100]mm/sec CNT100;
   1:  PR[GP1:91,1] = PR[GP1:90,1] + 48.995;
   1:  PR[GP1:91,2] = PR[GP1:90,2] + 33.154;
   1:L PR[91] R[100]mm/sec CNT100;
   1:  PR[GP1:91,1] = PR[GP1:90,1] + 42.694;
   1:  PR[GP1:91,2] = PR[GP1:90,2] + 34.228;
   1:L PR[91] R[100]mm/sec CNT100;
   1:  PR[GP1:91,1] = PR[GP1:90,1] + 36.303;
   1:  PR[GP1:91,2] = PR[GP1:90,2] + 34.112;
   1:L PR[91] R[100]mm/sec CNT100;
   1:  PR[GP1:91,1] = PR[GP1:90,1] + 36.245;
   1:  PR[GP1:91,2] = PR[GP1:90,2] + 34.105;
   1:L PR[91] R[100]mm/sec CNT100;
   1:  PR[GP1:91,1] = PR[GP1:90,1] + 29.988;
   1:  PR[GP1:91,2] = PR[GP1:90,2] + 32.803;
   1:L PR[91] R[100]mm/sec CNT100;
   1:  PR[GP1:91,1] = PR[GP1:90,1] + 24.081;
   1:  PR[GP1:91,2] = PR[GP1:90,2] + 30.361;
   1:L PR[91] R[100]mm/sec CNT100;
   1:  PR[GP1:91,1] = PR[GP1:90,1] + 24.030;
   1:  PR[GP1:91,2] = PR[GP1:90,2] + 30.334;
   1:L PR[91] R[100]mm/sec CNT100;
   1:  PR[GP1:91,1] = PR[GP1:90,1] + 18.680;
   1:  PR[GP1:91,2] = PR[GP1:90,2] + 26.836;
   1:L PR[91] R[100]mm/sec CNT100;
   1:  PR[GP1:91,1] = PR[GP1:90,1] + 14.073;
   1:  PR[GP1:91,2] = PR[GP1:90,2] + 22.406;
   1:L PR[91] R[100]mm/sec CNT100;
   1:  PR[GP1:91,1] = PR[GP1:90,1] + 14.035;
   1:  PR[GP1:91,2] = PR[GP1:90,2] + 22.362;
   1:L PR[91] R[100]mm/sec CNT100;
   1:  PR[GP1:91,1] = PR[GP1:90,1] + 10.332;
   1:  PR[GP1:91,2] = PR[GP1:90,2] + 17.152;
   1:L PR[91] R[100]mm/sec CNT100;
   1:  PR[GP1:91,1] = PR[GP1:90,1] + 7.662;
   1:  PR[GP1:91,2] = PR[GP1:90,2] + 11.344;
   1:L PR[91] R[100]mm/sec CNT100;
   1:  PR[GP1:91,1] = PR[GP1:90,1] + 7.643;
   1:  PR[GP1:91,2] = PR[GP1:90,2] + 11.290;
   1:L PR[91] R[100]mm/sec CNT100;
   1:  PR[GP1:91,1] = PR[GP1:90,1] + 6.066;
   1:  PR[GP1:91,2] = PR[GP1:90,2] + 4.956;
   1:L PR[91] R[100]mm/sec CNT100;
   1:  PR[GP1:91,1] = PR[GP1:90,1] + 4.236;
   1:  PR[GP1:91,2] = PR[GP1:90,2] + 1.651;
   1:L PR[91] R[100]mm/sec CNT100;
   1:  PR[GP1:91,1] = PR[GP1:90,1] + 0.667;
   1:  PR[GP1:91,2] = PR[GP1:90,2] + 0.328;
   1:L PR[91] R[100]mm/sec CNT100;
   1:  PR[GP1:91,1] = PR[GP1:90,1] + -0.454;
   1:L PR[91] R[100]mm/sec CNT100;
   1:  ! -- Layer/Ebene 14 -- !;
   1:  PR[91] = PR[90];
   1:  PR[GP1:91,1] = PR[GP1:90,1] + -3.983;
   1:  PR[GP1:91,2] = PR[GP1:90,2] + 1.652;
   1:  PR[GP1:91,3] = PR[GP1:90,3] + 8.845;
   1:L PR[91] R[100]mm/sec CNT100;
   1:  PR[GP1:91,1] = PR[GP1:90,1] + -5.628;
   1:  PR[GP1:91,2] = PR[GP1:90,2] + 4.623;
   1:L PR[91] R[100]mm/sec CNT100;
   1:  PR[GP1:91,1] = PR[GP1:90,1] + -6.111;
   1:  PR[GP1:91,2] = PR[GP1:90,2] + 5.392;
   1:L PR[91] R[100]mm/sec CNT100;
   1:  PR[GP1:91,1] = PR[GP1:90,1] + -5.943;
   1:  PR[GP1:91,2] = PR[GP1:90,2] + 5.486;
   1:L PR[91] R[100]mm/sec CNT100;
   1:  PR[GP1:91,1] = PR[GP1:90,1] + -7.284;
   1:  PR[GP1:91,2] = PR[GP1:90,2] + 10.871;
   1:L PR[91] R[100]mm/sec CNT100;
   1:  PR[GP1:91,1] = PR[GP1:90,1] + -7.543;
   1:  PR[GP1:91,2] = PR[GP1:90,2] + 11.653;
   1:L PR[91] R[100]mm/sec CNT100;
   1:  PR[GP1:91,1] = PR[GP1:90,1] + -10.033;
   1:  PR[GP1:91,2] = PR[GP1:90,2] + 17.069;
   1:L PR[91] R[100]mm/sec CNT100;
   1:  PR[GP1:91,1] = PR[GP1:90,1] + -13.500;
   1:  PR[GP1:91,2] = PR[GP1:90,2] + 21.947;
   1:L PR[91] R[100]mm/sec CNT100;
   1:  PR[GP1:91,1] = PR[GP1:90,1] + -13.976;
   1:  PR[GP1:91,2] = PR[GP1:90,2] + 22.571;
   1:L PR[91] R[100]mm/sec CNT100;
   1:  PR[GP1:91,1] = PR[GP1:90,1] + -18.285;
   1:  PR[GP1:91,2] = PR[GP1:90,2] + 26.715;
   1:L PR[91] R[100]mm/sec CNT100;
   1:  PR[GP1:91,1] = PR[GP1:90,1] + -23.942;
   1:  PR[GP1:91,2] = PR[GP1:90,2] + 30.419;
   1:L PR[91] R[100]mm/sec CNT100;
   1:  PR[GP1:91,1] = PR[GP1:90,1] + -29.489;
   1:  PR[GP1:91,2] = PR[GP1:90,2] + 32.713;
   1:L PR[91] R[100]mm/sec CNT100;
   1:  PR[GP1:91,1] = PR[GP1:90,1] + -35.435;
   1:  PR[GP1:91,2] = PR[GP1:90,2] + 33.950;
   1:L PR[91] R[100]mm/sec CNT100;
   1:  PR[GP1:91,1] = PR[GP1:90,1] + -36.096;
   1:  PR[GP1:91,2] = PR[GP1:90,2] + 34.121;
   1:L PR[91] R[100]mm/sec CNT100;
   1:  PR[GP1:91,1] = PR[GP1:90,1] + -42.146;
   1:  PR[GP1:91,2] = PR[GP1:90,2] + 34.231;
   1:L PR[91] R[100]mm/sec CNT100;
   1:  PR[GP1:91,1] = PR[GP1:90,1] + -42.743;
   1:  PR[GP1:91,2] = PR[GP1:90,2] + 34.186;
   1:L PR[91] R[100]mm/sec CNT100;
   1:  PR[GP1:91,1] = PR[GP1:90,1] + -48.752;
   1:  PR[GP1:91,2] = PR[GP1:90,2] + 33.162;
   1:L PR[91] R[100]mm/sec CNT100;
   1:  PR[GP1:91,1] = PR[GP1:90,1] + -54.478;
   1:  PR[GP1:91,2] = PR[GP1:90,2] + 31.035;
   1:L PR[91] R[100]mm/sec CNT100;
   1:  PR[GP1:91,1] = PR[GP1:90,1] + -54.989;
   1:  PR[GP1:91,2] = PR[GP1:90,2] + 30.815;
   1:L PR[91] R[100]mm/sec CNT100;
   1:  PR[GP1:91,1] = PR[GP1:90,1] + -60.218;
   1:  PR[GP1:91,2] = PR[GP1:90,2] + 27.662;
   1:L PR[91] R[100]mm/sec CNT100;
   1:  PR[GP1:91,1] = PR[GP1:90,1] + -65.186;
   1:  PR[GP1:91,2] = PR[GP1:90,2] + 23.213;
   1:L PR[91] R[100]mm/sec CNT100;
   1:  PR[GP1:91,1] = PR[GP1:90,1] + -68.903;
   1:  PR[GP1:91,2] = PR[GP1:90,2] + 18.366;
   1:L PR[91] R[100]mm/sec CNT100;
   1:  PR[GP1:91,1] = PR[GP1:90,1] + -71.685;
   1:  PR[GP1:91,2] = PR[GP1:90,2] + 12.854;
   1:L PR[91] R[100]mm/sec CNT100;
   1:  PR[GP1:91,1] = PR[GP1:90,1] + -71.922;
   1:  PR[GP1:91,2] = PR[GP1:90,2] + 12.419;
   1:L PR[91] R[100]mm/sec CNT100;
   1:  PR[GP1:91,1] = PR[GP1:90,1] + -73.613;
   1:  PR[GP1:91,2] = PR[GP1:90,2] + 6.548;
   1:L PR[91] R[100]mm/sec CNT100;
   1:  PR[GP1:91,1] = PR[GP1:90,1] + -74.191;
   1:  PR[GP1:91,2] = PR[GP1:90,2] + 0.380;
   1:L PR[91] R[100]mm/sec CNT100;
   1:  PR[GP1:91,1] = PR[GP1:90,1] + -74.270;
   1:  PR[GP1:91,2] = PR[GP1:90,2] + -0.094;
   1:L PR[91] R[100]mm/sec CNT100;
   1:  PR[GP1:91,1] = PR[GP1:90,1] + -73.697;
   1:  PR[GP1:91,2] = PR[GP1:90,2] + -6.208;
   1:L PR[91] R[100]mm/sec CNT100;
   1:  PR[GP1:91,1] = PR[GP1:90,1] + -73.619;
   1:  PR[GP1:91,2] = PR[GP1:90,2] + -6.671;
   1:L PR[91] R[100]mm/sec CNT100;
   1:  PR[GP1:91,1] = PR[GP1:90,1] + -71.919;
   1:  PR[GP1:91,2] = PR[GP1:90,2] + -12.572;
   1:L PR[91] R[100]mm/sec CNT100;
   1:  PR[GP1:91,1] = PR[GP1:90,1] + -69.142;
   1:  PR[GP1:91,2] = PR[GP1:90,2] + -18.075;
   1:L PR[91] R[100]mm/sec CNT100;
   1:  PR[GP1:91,1] = PR[GP1:90,1] + -68.909;
   1:  PR[GP1:91,2] = PR[GP1:90,2] + -18.502;
   1:L PR[91] R[100]mm/sec CNT100;
   1:  PR[GP1:91,1] = PR[GP1:90,1] + -65.186;
   1:  PR[GP1:91,2] = PR[GP1:90,2] + -23.357;
   1:L PR[91] R[100]mm/sec CNT100;
   1:  PR[GP1:91,1] = PR[GP1:90,1] + -60.218;
   1:  PR[GP1:91,2] = PR[GP1:90,2] + -27.806;
   1:L PR[91] R[100]mm/sec CNT100;
   1:  PR[GP1:91,1] = PR[GP1:90,1] + -55.002;
   1:  PR[GP1:91,2] = PR[GP1:90,2] + -30.951;
   1:L PR[91] R[100]mm/sec CNT100;
   1:  PR[GP1:91,1] = PR[GP1:90,1] + -49.224;
   1:  PR[GP1:91,2] = PR[GP1:90,2] + -33.098;
   1:L PR[91] R[100]mm/sec CNT100;
   1:  PR[GP1:91,1] = PR[GP1:90,1] + -48.736;
   1:  PR[GP1:91,2] = PR[GP1:90,2] + -33.309;
   1:L PR[91] R[100]mm/sec CNT100;
   1:  PR[GP1:91,1] = PR[GP1:90,1] + -42.743;
   1:  PR[GP1:91,2] = PR[GP1:90,2] + -34.330;
   1:L PR[91] R[100]mm/sec CNT100;
   1:  PR[GP1:91,1] = PR[GP1:90,1] + -42.146;
   1:  PR[GP1:91,2] = PR[GP1:90,2] + -34.375;
   1:L PR[91] R[100]mm/sec CNT100;
   1:  PR[GP1:91,1] = PR[GP1:90,1] + -36.081;
   1:  PR[GP1:91,2] = PR[GP1:90,2] + -34.265;
   1:L PR[91] R[100]mm/sec CNT100;
   1:  PR[GP1:91,1] = PR[GP1:90,1] + -30.130;
   1:  PR[GP1:91,2] = PR[GP1:90,2] + -33.027;
   1:L PR[91] R[100]mm/sec CNT100;
   1:  PR[GP1:91,1] = PR[GP1:90,1] + -29.503;
   1:  PR[GP1:91,2] = PR[GP1:90,2] + -32.863;
   1:L PR[91] R[100]mm/sec CNT100;
   1:  PR[GP1:91,1] = PR[GP1:90,1] + -23.942;
   1:  PR[GP1:91,2] = PR[GP1:90,2] + -30.563;
   1:L PR[91] R[100]mm/sec CNT100;
   1:  PR[GP1:91,1] = PR[GP1:90,1] + -18.285;
   1:  PR[GP1:91,2] = PR[GP1:90,2] + -26.859;
   1:L PR[91] R[100]mm/sec CNT100;
   1:  PR[GP1:91,1] = PR[GP1:90,1] + -13.984;
   1:  PR[GP1:91,2] = PR[GP1:90,2] + -22.722;
   1:L PR[91] R[100]mm/sec CNT100;
   1:  PR[GP1:91,1] = PR[GP1:90,1] + -10.488;
   1:  PR[GP1:91,2] = PR[GP1:90,2] + -17.803;
   1:L PR[91] R[100]mm/sec CNT100;
   1:  PR[GP1:91,1] = PR[GP1:90,1] + -10.028;
   1:  PR[GP1:91,2] = PR[GP1:90,2] + -17.204;
   1:L PR[91] R[100]mm/sec CNT100;
   1:  PR[GP1:91,1] = PR[GP1:90,1] + -7.543;
   1:  PR[GP1:91,2] = PR[GP1:90,2] + -11.797;
   1:L PR[91] R[100]mm/sec CNT100;
   1:  PR[GP1:91,1] = PR[GP1:90,1] + -7.284;
   1:  PR[GP1:91,2] = PR[GP1:90,2] + -11.015;
   1:L PR[91] R[100]mm/sec CNT100;
   1:  PR[GP1:91,1] = PR[GP1:90,1] + -5.941;
   1:  PR[GP1:91,2] = PR[GP1:90,2] + -5.624;
   1:L PR[91] R[100]mm/sec CNT100;
   1:  PR[GP1:91,1] = PR[GP1:90,1] + -6.076;
   1:  PR[GP1:91,2] = PR[GP1:90,2] + -5.545;
   1:L PR[91] R[100]mm/sec CNT100;
   1:  PR[GP1:91,1] = PR[GP1:90,1] + -4.116;
   1:  PR[GP1:91,2] = PR[GP1:90,2] + -1.992;
   1:L PR[91] R[100]mm/sec CNT100;
   1:  PR[GP1:91,1] = PR[GP1:90,1] + -3.966;
   1:  PR[GP1:91,2] = PR[GP1:90,2] + -1.829;
   1:L PR[91] R[100]mm/sec CNT100;
   1:  PR[GP1:91,1] = PR[GP1:90,1] + -3.762;
   1:  PR[GP1:91,2] = PR[GP1:90,2] + -1.689;
   1:L PR[91] R[100]mm/sec CNT100;
   1:  PR[GP1:91,1] = PR[GP1:90,1] + -0.681;
   1:  PR[GP1:91,2] = PR[GP1:90,2] + -0.546;
   1:L PR[91] R[100]mm/sec CNT100;
   1:  PR[GP1:91,1] = PR[GP1:90,1] + -0.403;
   1:  PR[GP1:91,2] = PR[GP1:90,2] + -0.472;
   1:L PR[91] R[100]mm/sec CNT100;
   1:  PR[GP1:91,1] = PR[GP1:90,1] + 0.646;
   1:L PR[91] R[100]mm/sec CNT100;
   1:  PR[GP1:91,1] = PR[GP1:90,1] + 4.197;
   1:  PR[GP1:91,2] = PR[GP1:90,2] + -1.796;
   1:L PR[91] R[100]mm/sec CNT100;
   1:  PR[GP1:91,1] = PR[GP1:90,1] + 5.842;
   1:  PR[GP1:91,2] = PR[GP1:90,2] + -4.767;
   1:L PR[91] R[100]mm/sec CNT100;
   1:  PR[GP1:91,1] = PR[GP1:90,1] + 6.322;
   1:  PR[GP1:91,2] = PR[GP1:90,2] + -5.534;
   1:L PR[91] R[100]mm/sec CNT100;
   1:  PR[GP1:91,1] = PR[GP1:90,1] + 6.156;
   1:  PR[GP1:91,2] = PR[GP1:90,2] + -5.629;
   1:L PR[91] R[100]mm/sec CNT100;
   1:  PR[GP1:91,1] = PR[GP1:90,1] + 7.497;
   1:  PR[GP1:91,2] = PR[GP1:90,2] + -11.015;
   1:L PR[91] R[100]mm/sec CNT100;
   1:  PR[GP1:91,1] = PR[GP1:90,1] + 7.756;
   1:  PR[GP1:91,2] = PR[GP1:90,2] + -11.797;
   1:L PR[91] R[100]mm/sec CNT100;
   1:  PR[GP1:91,1] = PR[GP1:90,1] + 10.246;
   1:  PR[GP1:91,2] = PR[GP1:90,2] + -17.213;
   1:L PR[91] R[100]mm/sec CNT100;
   1:  PR[GP1:91,1] = PR[GP1:90,1] + 13.713;
   1:  PR[GP1:91,2] = PR[GP1:90,2] + -22.091;
   1:L PR[91] R[100]mm/sec CNT100;
   1:  PR[GP1:91,1] = PR[GP1:90,1] + 14.190;
   1:  PR[GP1:91,2] = PR[GP1:90,2] + -22.715;
   1:L PR[91] R[100]mm/sec CNT100;
   1:  PR[GP1:91,1] = PR[GP1:90,1] + 18.498;
   1:  PR[GP1:91,2] = PR[GP1:90,2] + -26.859;
   1:L PR[91] R[100]mm/sec CNT100;
   1:  PR[GP1:91,1] = PR[GP1:90,1] + 24.155;
   1:  PR[GP1:91,2] = PR[GP1:90,2] + -30.563;
   1:L PR[91] R[100]mm/sec CNT100;
   1:  PR[GP1:91,1] = PR[GP1:90,1] + 29.702;
   1:  PR[GP1:91,2] = PR[GP1:90,2] + -32.857;
   1:L PR[91] R[100]mm/sec CNT100;
   1:  PR[GP1:91,1] = PR[GP1:90,1] + 35.648;
   1:  PR[GP1:91,2] = PR[GP1:90,2] + -34.094;
   1:L PR[91] R[100]mm/sec CNT100;
   1:  PR[GP1:91,1] = PR[GP1:90,1] + 36.309;
   1:  PR[GP1:91,2] = PR[GP1:90,2] + -34.265;
   1:L PR[91] R[100]mm/sec CNT100;
   1:  PR[GP1:91,1] = PR[GP1:90,1] + 42.359;
   1:  PR[GP1:91,2] = PR[GP1:90,2] + -34.375;
   1:L PR[91] R[100]mm/sec CNT100;
   1:  PR[GP1:91,1] = PR[GP1:90,1] + 42.956;
   1:  PR[GP1:91,2] = PR[GP1:90,2] + -34.330;
   1:L PR[91] R[100]mm/sec CNT100;
   1:  PR[GP1:91,1] = PR[GP1:90,1] + 48.965;
   1:  PR[GP1:91,2] = PR[GP1:90,2] + -33.306;
   1:L PR[91] R[100]mm/sec CNT100;
   1:  PR[GP1:91,1] = PR[GP1:90,1] + 54.691;
   1:  PR[GP1:91,2] = PR[GP1:90,2] + -31.179;
   1:L PR[91] R[100]mm/sec CNT100;
   1:  PR[GP1:91,1] = PR[GP1:90,1] + 55.202;
   1:  PR[GP1:91,2] = PR[GP1:90,2] + -30.959;
   1:L PR[91] R[100]mm/sec CNT100;
   1:  PR[GP1:91,1] = PR[GP1:90,1] + 60.431;
   1:  PR[GP1:91,2] = PR[GP1:90,2] + -27.806;
   1:L PR[91] R[100]mm/sec CNT100;
   1:  PR[GP1:91,1] = PR[GP1:90,1] + 65.399;
   1:  PR[GP1:91,2] = PR[GP1:90,2] + -23.357;
   1:L PR[91] R[100]mm/sec CNT100;
   1:  PR[GP1:91,1] = PR[GP1:90,1] + 69.116;
   1:  PR[GP1:91,2] = PR[GP1:90,2] + -18.510;
   1:L PR[91] R[100]mm/sec CNT100;
   1:  PR[GP1:91,1] = PR[GP1:90,1] + 71.898;
   1:  PR[GP1:91,2] = PR[GP1:90,2] + -12.998;
   1:L PR[91] R[100]mm/sec CNT100;
   1:  PR[GP1:91,1] = PR[GP1:90,1] + 72.135;
   1:  PR[GP1:91,2] = PR[GP1:90,2] + -12.563;
   1:L PR[91] R[100]mm/sec CNT100;
   1:  PR[GP1:91,1] = PR[GP1:90,1] + 73.826;
   1:  PR[GP1:91,2] = PR[GP1:90,2] + -6.693;
   1:L PR[91] R[100]mm/sec CNT100;
   1:  PR[GP1:91,1] = PR[GP1:90,1] + 74.404;
   1:  PR[GP1:91,2] = PR[GP1:90,2] + -0.524;
   1:L PR[91] R[100]mm/sec CNT100;
   1:  PR[GP1:91,1] = PR[GP1:90,1] + 74.483;
   1:  PR[GP1:91,2] = PR[GP1:90,2] + -0.050;
   1:L PR[91] R[100]mm/sec CNT100;
   1:  PR[GP1:91,1] = PR[GP1:90,1] + 73.910;
   1:  PR[GP1:91,2] = PR[GP1:90,2] + 6.064;
   1:L PR[91] R[100]mm/sec CNT100;
   1:  PR[GP1:91,1] = PR[GP1:90,1] + 73.832;
   1:  PR[GP1:91,2] = PR[GP1:90,2] + 6.527;
   1:L PR[91] R[100]mm/sec CNT100;
   1:  PR[GP1:91,1] = PR[GP1:90,1] + 72.133;
   1:  PR[GP1:91,2] = PR[GP1:90,2] + 12.428;
   1:L PR[91] R[100]mm/sec CNT100;
   1:  PR[GP1:91,1] = PR[GP1:90,1] + 69.355;
   1:  PR[GP1:91,2] = PR[GP1:90,2] + 17.931;
   1:L PR[91] R[100]mm/sec CNT100;
   1:  PR[GP1:91,1] = PR[GP1:90,1] + 69.122;
   1:  PR[GP1:91,2] = PR[GP1:90,2] + 18.358;
   1:L PR[91] R[100]mm/sec CNT100;
   1:  PR[GP1:91,1] = PR[GP1:90,1] + 65.399;
   1:  PR[GP1:91,2] = PR[GP1:90,2] + 23.213;
   1:L PR[91] R[100]mm/sec CNT100;
   1:  PR[GP1:91,1] = PR[GP1:90,1] + 60.431;
   1:  PR[GP1:91,2] = PR[GP1:90,2] + 27.662;
   1:L PR[91] R[100]mm/sec CNT100;
   1:  PR[GP1:91,1] = PR[GP1:90,1] + 55.215;
   1:  PR[GP1:91,2] = PR[GP1:90,2] + 30.807;
   1:L PR[91] R[100]mm/sec CNT100;
   1:  PR[GP1:91,1] = PR[GP1:90,1] + 49.437;
   1:  PR[GP1:91,2] = PR[GP1:90,2] + 32.954;
   1:L PR[91] R[100]mm/sec CNT100;
   1:  PR[GP1:91,1] = PR[GP1:90,1] + 48.949;
   1:  PR[GP1:91,2] = PR[GP1:90,2] + 33.165;
   1:L PR[91] R[100]mm/sec CNT100;
   1:  PR[GP1:91,1] = PR[GP1:90,1] + 42.956;
   1:  PR[GP1:91,2] = PR[GP1:90,2] + 34.186;
   1:L PR[91] R[100]mm/sec CNT100;
   1:  PR[GP1:91,1] = PR[GP1:90,1] + 42.359;
   1:  PR[GP1:91,2] = PR[GP1:90,2] + 34.231;
   1:L PR[91] R[100]mm/sec CNT100;
   1:  PR[GP1:91,1] = PR[GP1:90,1] + 36.294;
   1:  PR[GP1:91,2] = PR[GP1:90,2] + 34.121;
   1:L PR[91] R[100]mm/sec CNT100;
   1:  PR[GP1:91,1] = PR[GP1:90,1] + 30.343;
   1:  PR[GP1:91,2] = PR[GP1:90,2] + 32.883;
   1:L PR[91] R[100]mm/sec CNT100;
   1:  PR[GP1:91,1] = PR[GP1:90,1] + 29.716;
   1:  PR[GP1:91,2] = PR[GP1:90,2] + 32.719;
   1:L PR[91] R[100]mm/sec CNT100;
   1:  PR[GP1:91,1] = PR[GP1:90,1] + 24.155;
   1:  PR[GP1:91,2] = PR[GP1:90,2] + 30.419;
   1:L PR[91] R[100]mm/sec CNT100;
   1:  PR[GP1:91,1] = PR[GP1:90,1] + 18.498;
   1:  PR[GP1:91,2] = PR[GP1:90,2] + 26.715;
   1:L PR[91] R[100]mm/sec CNT100;
   1:  PR[GP1:91,1] = PR[GP1:90,1] + 14.197;
   1:  PR[GP1:91,2] = PR[GP1:90,2] + 22.578;
   1:L PR[91] R[100]mm/sec CNT100;
   1:  PR[GP1:91,1] = PR[GP1:90,1] + 10.701;
   1:  PR[GP1:91,2] = PR[GP1:90,2] + 17.659;
   1:L PR[91] R[100]mm/sec CNT100;
   1:  PR[GP1:91,1] = PR[GP1:90,1] + 10.242;
   1:  PR[GP1:91,2] = PR[GP1:90,2] + 17.059;
   1:L PR[91] R[100]mm/sec CNT100;
   1:  PR[GP1:91,1] = PR[GP1:90,1] + 7.756;
   1:  PR[GP1:91,2] = PR[GP1:90,2] + 11.653;
   1:L PR[91] R[100]mm/sec CNT100;
   1:  PR[GP1:91,1] = PR[GP1:90,1] + 7.497;
   1:  PR[GP1:91,2] = PR[GP1:90,2] + 10.871;
   1:L PR[91] R[100]mm/sec CNT100;
   1:  PR[GP1:91,1] = PR[GP1:90,1] + 6.155;
   1:  PR[GP1:91,2] = PR[GP1:90,2] + 5.482;
   1:L PR[91] R[100]mm/sec CNT100;
   1:  PR[GP1:91,1] = PR[GP1:90,1] + 6.290;
   1:  PR[GP1:91,2] = PR[GP1:90,2] + 5.403;
   1:L PR[91] R[100]mm/sec CNT100;
   1:  PR[GP1:91,1] = PR[GP1:90,1] + 4.329;
   1:  PR[GP1:91,2] = PR[GP1:90,2] + 1.848;
   1:L PR[91] R[100]mm/sec CNT100;
   1:  PR[GP1:91,1] = PR[GP1:90,1] + 4.179;
   1:  PR[GP1:91,2] = PR[GP1:90,2] + 1.685;
   1:L PR[91] R[100]mm/sec CNT100;
   1:  PR[GP1:91,1] = PR[GP1:90,1] + 3.976;
   1:  PR[GP1:91,2] = PR[GP1:90,2] + 1.545;
   1:L PR[91] R[100]mm/sec CNT100;
   1:  PR[GP1:91,1] = PR[GP1:90,1] + 0.894;
   1:  PR[GP1:91,2] = PR[GP1:90,2] + 0.402;
   1:L PR[91] R[100]mm/sec CNT100;
   1:  PR[GP1:91,1] = PR[GP1:90,1] + 0.616;
   1:  PR[GP1:91,2] = PR[GP1:90,2] + 0.328;
   1:L PR[91] R[100]mm/sec CNT100;
   1:  PR[GP1:91,1] = PR[GP1:90,1] + -0.433;
   1:L PR[91] R[100]mm/sec CNT100;
   1:  ! -- Layer/Ebene 15 -- !;
   1:  PR[91] = PR[90];
   1:  PR[GP1:91,1] = PR[GP1:90,1] + -2.594;
   1:  PR[GP1:91,2] = PR[GP1:90,2] + 1.138;
   1:  PR[GP1:91,3] = PR[GP1:90,3] + 9.455;
   1:L PR[91] R[100]mm/sec CNT100;
   1:  PR[GP1:91,1] = PR[GP1:90,1] + -3.035;
   1:  PR[GP1:91,2] = PR[GP1:90,2] + 1.314;
   1:L PR[91] R[100]mm/sec CNT100;
   1:  PR[GP1:91,1] = PR[GP1:90,1] + -3.078;
   1:  PR[GP1:91,2] = PR[GP1:90,2] + 1.316;
   1:L PR[91] R[100]mm/sec CNT100;
   1:  PR[GP1:91,1] = PR[GP1:90,1] + -3.942;
   1:  PR[GP1:91,2] = PR[GP1:90,2] + 1.658;
   1:L PR[91] R[100]mm/sec CNT100;
   1:  PR[GP1:91,1] = PR[GP1:90,1] + -5.427;
   1:  PR[GP1:91,2] = PR[GP1:90,2] + 4.341;
   1:L PR[91] R[100]mm/sec CNT100;
   1:  PR[GP1:91,1] = PR[GP1:90,1] + -6.086;
   1:  PR[GP1:91,2] = PR[GP1:90,2] + 5.392;
   1:L PR[91] R[100]mm/sec CNT100;
   1:  PR[GP1:91,1] = PR[GP1:90,1] + -5.898;
   1:  PR[GP1:91,2] = PR[GP1:90,2] + 5.498;
   1:L PR[91] R[100]mm/sec CNT100;
   1:  PR[GP1:91,1] = PR[GP1:90,1] + -7.101;
   1:  PR[GP1:91,2] = PR[GP1:90,2] + 10.330;
   1:L PR[91] R[100]mm/sec CNT100;
   1:  PR[GP1:91,1] = PR[GP1:90,1] + -7.673;
   1:  PR[GP1:91,2] = PR[GP1:90,2] + 12.056;
   1:L PR[91] R[100]mm/sec CNT100;
   1:  PR[GP1:91,1] = PR[GP1:90,1] + -9.936;
   1:  PR[GP1:91,2] = PR[GP1:90,2] + 16.976;
   1:L PR[91] R[100]mm/sec CNT100;
   1:  PR[GP1:91,1] = PR[GP1:90,1] + -13.087;
   1:  PR[GP1:91,2] = PR[GP1:90,2] + 21.409;
   1:L PR[91] R[100]mm/sec CNT100;
   1:  PR[GP1:91,1] = PR[GP1:90,1] + -14.140;
   1:  PR[GP1:91,2] = PR[GP1:90,2] + 22.788;
   1:L PR[91] R[100]mm/sec CNT100;
   1:  PR[GP1:91,1] = PR[GP1:90,1] + -18.081;
   1:  PR[GP1:91,2] = PR[GP1:90,2] + 26.578;
   1:L PR[91] R[100]mm/sec CNT100;
   1:  PR[GP1:91,1] = PR[GP1:90,1] + -24.055;
   1:  PR[GP1:91,2] = PR[GP1:90,2] + 30.497;
   1:L PR[91] R[100]mm/sec CNT100;
   1:  PR[GP1:91,1] = PR[GP1:90,1] + -29.166;
   1:  PR[GP1:91,2] = PR[GP1:90,2] + 32.611;
   1:L PR[91] R[100]mm/sec CNT100;
   1:  PR[GP1:91,1] = PR[GP1:90,1] + -34.650;
   1:  PR[GP1:91,2] = PR[GP1:90,2] + 33.752;
   1:L PR[91] R[100]mm/sec CNT100;
   1:  PR[GP1:91,1] = PR[GP1:90,1] + -36.119;
   1:  PR[GP1:91,2] = PR[GP1:90,2] + 34.132;
   1:L PR[91] R[100]mm/sec CNT100;
   1:  PR[GP1:91,1] = PR[GP1:90,1] + -41.736;
   1:  PR[GP1:91,2] = PR[GP1:90,2] + 34.234;
   1:L PR[91] R[100]mm/sec CNT100;
   1:  PR[GP1:91,1] = PR[GP1:90,1] + -43.071;
   1:  PR[GP1:91,2] = PR[GP1:90,2] + 34.134;
   1:L PR[91] R[100]mm/sec CNT100;
   1:  PR[GP1:91,1] = PR[GP1:90,1] + -48.687;
   1:  PR[GP1:91,2] = PR[GP1:90,2] + 33.177;
   1:L PR[91] R[100]mm/sec CNT100;
   1:  PR[GP1:91,1] = PR[GP1:90,1] + -54.039;
   1:  PR[GP1:91,2] = PR[GP1:90,2] + 31.189;
   1:L PR[91] R[100]mm/sec CNT100;
   1:  PR[GP1:91,1] = PR[GP1:90,1] + -55.184;
   1:  PR[GP1:91,2] = PR[GP1:90,2] + 30.695;
   1:L PR[91] R[100]mm/sec CNT100;
   1:  PR[GP1:91,1] = PR[GP1:90,1] + -60.094;
   1:  PR[GP1:91,2] = PR[GP1:90,2] + 27.734;
   1:L PR[91] R[100]mm/sec CNT100;
   1:  PR[GP1:91,1] = PR[GP1:90,1] + -65.267;
   1:  PR[GP1:91,2] = PR[GP1:90,2] + 23.094;
   1:L PR[91] R[100]mm/sec CNT100;
   1:  PR[GP1:91,1] = PR[GP1:90,1] + -68.769;
   1:  PR[GP1:91,2] = PR[GP1:90,2] + 18.527;
   1:L PR[91] R[100]mm/sec CNT100;
   1:  PR[GP1:91,1] = PR[GP1:90,1] + -71.392;
   1:  PR[GP1:91,2] = PR[GP1:90,2] + 13.331;
   1:L PR[91] R[100]mm/sec CNT100;
   1:  PR[GP1:91,1] = PR[GP1:90,1] + -71.927;
   1:  PR[GP1:91,2] = PR[GP1:90,2] + 12.347;
   1:L PR[91] R[100]mm/sec CNT100;
   1:  PR[GP1:91,1] = PR[GP1:90,1] + -73.523;
   1:  PR[GP1:91,2] = PR[GP1:90,2] + 6.806;
   1:L PR[91] R[100]mm/sec CNT100;
   1:  PR[GP1:91,1] = PR[GP1:90,1] + -74.070;
   1:  PR[GP1:91,2] = PR[GP1:90,2] + 0.977;
   1:L PR[91] R[100]mm/sec CNT100;
   1:  PR[GP1:91,1] = PR[GP1:90,1] + -74.248;
   1:  PR[GP1:91,2] = PR[GP1:90,2] + -0.094;
   1:L PR[91] R[100]mm/sec CNT100;
   1:  PR[GP1:91,1] = PR[GP1:90,1] + -73.706;
   1:  PR[GP1:91,2] = PR[GP1:90,2] + -5.880;
   1:L PR[91] R[100]mm/sec CNT100;
   1:  PR[GP1:91,1] = PR[GP1:90,1] + -73.530;
   1:  PR[GP1:91,2] = PR[GP1:90,2] + -6.928;
   1:L PR[91] R[100]mm/sec CNT100;
   1:  PR[GP1:91,1] = PR[GP1:90,1] + -71.925;
   1:  PR[GP1:91,2] = PR[GP1:90,2] + -12.500;
   1:L PR[91] R[100]mm/sec CNT100;
   1:  PR[GP1:91,1] = PR[GP1:90,1] + -69.301;
   1:  PR[GP1:91,2] = PR[GP1:90,2] + -17.699;
   1:L PR[91] R[100]mm/sec CNT100;
   1:  PR[GP1:91,1] = PR[GP1:90,1] + -68.775;
   1:  PR[GP1:91,2] = PR[GP1:90,2] + -18.664;
   1:L PR[91] R[100]mm/sec CNT100;
   1:  PR[GP1:91,1] = PR[GP1:90,1] + -65.267;
   1:  PR[GP1:91,2] = PR[GP1:90,2] + -23.238;
   1:L PR[91] R[100]mm/sec CNT100;
   1:  PR[GP1:91,1] = PR[GP1:90,1] + -60.094;
   1:  PR[GP1:91,2] = PR[GP1:90,2] + -27.878;
   1:L PR[91] R[100]mm/sec CNT100;
   1:  PR[GP1:91,1] = PR[GP1:90,1] + -55.197;
   1:  PR[GP1:91,2] = PR[GP1:90,2] + -30.831;
   1:L PR[91] R[100]mm/sec CNT100;
   1:  PR[GP1:91,1] = PR[GP1:90,1] + -49.768;
   1:  PR[GP1:91,2] = PR[GP1:90,2] + -32.848;
   1:L PR[91] R[100]mm/sec CNT100;
   1:  PR[GP1:91,1] = PR[GP1:90,1] + -48.671;
   1:  PR[GP1:91,2] = PR[GP1:90,2] + -33.324;
   1:L PR[91] R[100]mm/sec CNT100;
   1:  PR[GP1:91,1] = PR[GP1:90,1] + -43.071;
   1:  PR[GP1:91,2] = PR[GP1:90,2] + -34.278;
   1:L PR[91] R[100]mm/sec CNT100;
   1:  PR[GP1:91,1] = PR[GP1:90,1] + -41.736;
   1:  PR[GP1:91,2] = PR[GP1:90,2] + -34.378;
   1:L PR[91] R[100]mm/sec CNT100;
   1:  PR[GP1:91,1] = PR[GP1:90,1] + -36.105;
   1:  PR[GP1:91,2] = PR[GP1:90,2] + -34.276;
   1:L PR[91] R[100]mm/sec CNT100;
   1:  PR[GP1:91,1] = PR[GP1:90,1] + -30.578;
   1:  PR[GP1:91,2] = PR[GP1:90,2] + -33.126;
   1:L PR[91] R[100]mm/sec CNT100;
   1:  PR[GP1:91,1] = PR[GP1:90,1] + -29.180;
   1:  PR[GP1:91,2] = PR[GP1:90,2] + -32.760;
   1:L PR[91] R[100]mm/sec CNT100;
   1:  PR[GP1:91,1] = PR[GP1:90,1] + -24.055;
   1:  PR[GP1:91,2] = PR[GP1:90,2] + -30.641;
   1:L PR[91] R[100]mm/sec CNT100;
   1:  PR[GP1:91,1] = PR[GP1:90,1] + -18.080;
   1:  PR[GP1:91,2] = PR[GP1:90,2] + -26.722;
   1:L PR[91] R[100]mm/sec CNT100;
   1:  PR[GP1:91,1] = PR[GP1:90,1] + -14.148;
   1:  PR[GP1:91,2] = PR[GP1:90,2] + -22.940;
   1:L PR[91] R[100]mm/sec CNT100;
   1:  PR[GP1:91,1] = PR[GP1:90,1] + -10.948;
   1:  PR[GP1:91,2] = PR[GP1:90,2] + -18.438;
   1:L PR[91] R[100]mm/sec CNT100;
   1:  PR[GP1:91,1] = PR[GP1:90,1] + -9.931;
   1:  PR[GP1:91,2] = PR[GP1:90,2] + -17.110;
   1:L PR[91] R[100]mm/sec CNT100;
   1:  PR[GP1:91,1] = PR[GP1:90,1] + -7.673;
   1:  PR[GP1:91,2] = PR[GP1:90,2] + -12.200;
   1:L PR[91] R[100]mm/sec CNT100;
   1:  PR[GP1:91,1] = PR[GP1:90,1] + -7.102;
   1:  PR[GP1:91,2] = PR[GP1:90,2] + -10.474;
   1:L PR[91] R[100]mm/sec CNT100;
   1:  PR[GP1:91,1] = PR[GP1:90,1] + -5.897;
   1:  PR[GP1:91,2] = PR[GP1:90,2] + -5.636;
   1:L PR[91] R[100]mm/sec CNT100;
   1:  PR[GP1:91,1] = PR[GP1:90,1] + -6.051;
   1:  PR[GP1:91,2] = PR[GP1:90,2] + -5.546;
   1:L PR[91] R[100]mm/sec CNT100;
   1:  PR[GP1:91,1] = PR[GP1:90,1] + -4.139;
   1:  PR[GP1:91,2] = PR[GP1:90,2] + -2.065;
   1:L PR[91] R[100]mm/sec CNT100;
   1:  PR[GP1:91,1] = PR[GP1:90,1] + -3.926;
   1:  PR[GP1:91,2] = PR[GP1:90,2] + -1.834;
   1:L PR[91] R[100]mm/sec CNT100;
   1:  PR[GP1:91,1] = PR[GP1:90,1] + -3.624;
   1:  PR[GP1:91,2] = PR[GP1:90,2] + -1.626;
   1:L PR[91] R[100]mm/sec CNT100;
   1:  PR[GP1:91,1] = PR[GP1:90,1] + -0.854;
   1:  PR[GP1:91,2] = PR[GP1:90,2] + -0.599;
   1:L PR[91] R[100]mm/sec CNT100;
   1:  PR[GP1:91,1] = PR[GP1:90,1] + -0.378;
   1:  PR[GP1:91,2] = PR[GP1:90,2] + -0.472;
   1:L PR[91] R[100]mm/sec CNT100;
   1:  PR[GP1:91,1] = PR[GP1:90,1] + 0.622;
   1:L PR[91] R[100]mm/sec CNT100;
   1:  PR[GP1:91,1] = PR[GP1:90,1] + 2.807;
   1:  PR[GP1:91,2] = PR[GP1:90,2] + -1.282;
   1:L PR[91] R[100]mm/sec CNT100;
   1:  PR[GP1:91,1] = PR[GP1:90,1] + 3.248;
   1:  PR[GP1:91,2] = PR[GP1:90,2] + -1.458;
   1:L PR[91] R[100]mm/sec CNT100;
   1:  PR[GP1:91,1] = PR[GP1:90,1] + 3.291;
   1:  PR[GP1:91,2] = PR[GP1:90,2] + -1.460;
   1:L PR[91] R[100]mm/sec CNT100;
   1:  PR[GP1:91,1] = PR[GP1:90,1] + 4.155;
   1:  PR[GP1:91,2] = PR[GP1:90,2] + -1.802;
   1:L PR[91] R[100]mm/sec CNT100;
   1:  PR[GP1:91,1] = PR[GP1:90,1] + 5.641;
   1:  PR[GP1:91,2] = PR[GP1:90,2] + -4.485;
   1:L PR[91] R[100]mm/sec CNT100;
   1:  PR[GP1:91,1] = PR[GP1:90,1] + 6.298;
   1:  PR[GP1:91,2] = PR[GP1:90,2] + -5.534;
   1:L PR[91] R[100]mm/sec CNT100;
   1:  PR[GP1:91,1] = PR[GP1:90,1] + 6.111;
   1:  PR[GP1:91,2] = PR[GP1:90,2] + -5.640;
   1:L PR[91] R[100]mm/sec CNT100;
   1:  PR[GP1:91,1] = PR[GP1:90,1] + 7.315;
   1:  PR[GP1:91,2] = PR[GP1:90,2] + -10.474;
   1:L PR[91] R[100]mm/sec CNT100;
   1:  PR[GP1:91,1] = PR[GP1:90,1] + 7.887;
   1:  PR[GP1:91,2] = PR[GP1:90,2] + -12.199;
   1:L PR[91] R[100]mm/sec CNT100;
   1:  PR[GP1:91,1] = PR[GP1:90,1] + 10.149;
   1:  PR[GP1:91,2] = PR[GP1:90,2] + -17.119;
   1:L PR[91] R[100]mm/sec CNT100;
   1:  PR[GP1:91,1] = PR[GP1:90,1] + 13.300;
   1:  PR[GP1:91,2] = PR[GP1:90,2] + -21.553;
   1:L PR[91] R[100]mm/sec CNT100;
   1:  PR[GP1:91,1] = PR[GP1:90,1] + 14.353;
   1:  PR[GP1:91,2] = PR[GP1:90,2] + -22.932;
   1:L PR[91] R[100]mm/sec CNT100;
   1:  PR[GP1:91,1] = PR[GP1:90,1] + 18.293;
   1:  PR[GP1:91,2] = PR[GP1:90,2] + -26.722;
   1:L PR[91] R[100]mm/sec CNT100;
   1:  PR[GP1:91,1] = PR[GP1:90,1] + 24.268;
   1:  PR[GP1:91,2] = PR[GP1:90,2] + -30.641;
   1:L PR[91] R[100]mm/sec CNT100;
   1:  PR[GP1:91,1] = PR[GP1:90,1] + 29.379;
   1:  PR[GP1:91,2] = PR[GP1:90,2] + -32.754;
   1:L PR[91] R[100]mm/sec CNT100;
   1:  PR[GP1:91,1] = PR[GP1:90,1] + 34.863;
   1:  PR[GP1:91,2] = PR[GP1:90,2] + -33.895;
   1:L PR[91] R[100]mm/sec CNT100;
   1:  PR[GP1:91,1] = PR[GP1:90,1] + 36.332;
   1:  PR[GP1:91,2] = PR[GP1:90,2] + -34.276;
   1:L PR[91] R[100]mm/sec CNT100;
   1:  PR[GP1:91,1] = PR[GP1:90,1] + 41.949;
   1:  PR[GP1:91,2] = PR[GP1:90,2] + -34.378;
   1:L PR[91] R[100]mm/sec CNT100;
   1:  PR[GP1:91,1] = PR[GP1:90,1] + 43.284;
   1:  PR[GP1:91,2] = PR[GP1:90,2] + -34.278;
   1:L PR[91] R[100]mm/sec CNT100;
   1:  PR[GP1:91,1] = PR[GP1:90,1] + 48.900;
   1:  PR[GP1:91,2] = PR[GP1:90,2] + -33.321;
   1:L PR[91] R[100]mm/sec CNT100;
   1:  PR[GP1:91,1] = PR[GP1:90,1] + 54.252;
   1:  PR[GP1:91,2] = PR[GP1:90,2] + -31.333;
   1:L PR[91] R[100]mm/sec CNT100;
   1:  PR[GP1:91,1] = PR[GP1:90,1] + 55.397;
   1:  PR[GP1:91,2] = PR[GP1:90,2] + -30.839;
   1:L PR[91] R[100]mm/sec CNT100;
   1:  PR[GP1:91,1] = PR[GP1:90,1] + 60.307;
   1:  PR[GP1:91,2] = PR[GP1:90,2] + -27.879;
   1:L PR[91] R[100]mm/sec CNT100;
   1:  PR[GP1:91,1] = PR[GP1:90,1] + 65.480;
   1:  PR[GP1:91,2] = PR[GP1:90,2] + -23.238;
   1:L PR[91] R[100]mm/sec CNT100;
   1:  PR[GP1:91,1] = PR[GP1:90,1] + 68.983;
   1:  PR[GP1:91,2] = PR[GP1:90,2] + -18.671;
   1:L PR[91] R[100]mm/sec CNT100;
   1:  PR[GP1:91,1] = PR[GP1:90,1] + 71.605;
   1:  PR[GP1:91,2] = PR[GP1:90,2] + -13.475;
   1:L PR[91] R[100]mm/sec CNT100;
   1:  PR[GP1:91,1] = PR[GP1:90,1] + 72.141;
   1:  PR[GP1:91,2] = PR[GP1:90,2] + -12.492;
   1:L PR[91] R[100]mm/sec CNT100;
   1:  PR[GP1:91,1] = PR[GP1:90,1] + 73.737;
   1:  PR[GP1:91,2] = PR[GP1:90,2] + -6.950;
   1:L PR[91] R[100]mm/sec CNT100;
   1:  PR[GP1:91,1] = PR[GP1:90,1] + 74.283;
   1:  PR[GP1:91,2] = PR[GP1:90,2] + -1.122;
   1:L PR[91] R[100]mm/sec CNT100;
   1:  PR[GP1:91,1] = PR[GP1:90,1] + 74.462;
   1:  PR[GP1:91,2] = PR[GP1:90,2] + -0.050;
   1:L PR[91] R[100]mm/sec CNT100;
   1:  PR[GP1:91,1] = PR[GP1:90,1] + 73.919;
   1:  PR[GP1:91,2] = PR[GP1:90,2] + 5.736;
   1:L PR[91] R[100]mm/sec CNT100;
   1:  PR[GP1:91,1] = PR[GP1:90,1] + 73.743;
   1:  PR[GP1:91,2] = PR[GP1:90,2] + 6.785;
   1:L PR[91] R[100]mm/sec CNT100;
   1:  PR[GP1:91,1] = PR[GP1:90,1] + 72.138;
   1:  PR[GP1:91,2] = PR[GP1:90,2] + 12.357;
   1:L PR[91] R[100]mm/sec CNT100;
   1:  PR[GP1:91,1] = PR[GP1:90,1] + 69.515;
